// TwinCAT 3 PLC project MasterController
// ProgramVersion: 3.1.4024.0
// libraries:
//   Tc2_EtherCAT, * (Beckhoff Automation GmbH)
//   Tc2_Math, * (Beckhoff Automation GmbH)
//   Tc2_Standard, * (Beckhoff Automation GmbH)
//   Tc2_System, * (Beckhoff Automation GmbH)
//   Tc2_Utilities, * (Beckhoff Automation GmbH)
//   Tc3_Module, * (Beckhoff Automation GmbH)
// project tree:
//   AgiMaths/Frames/ DHTrans.TcPOU (not stored), invFrame.TcPOU (not stored), rotX.TcPOU (not stored), rotY.TcPOU (not stored), rotZ.TcPOU (not stored), transform.TcPOU (not stored)
//   AgiMaths/MatrixLib/ angAxis2Rot.TcPOU (not stored), cross.TcPOU (not stored), Det5.TcPOU (not stored), Det6.TcPOU (not stored), Det7.TcPOU (not stored), invMat6.TcPOU (not stored), invMat6Old.TcPOU (not stored), invMat3.TcPOU (not stored), invMat7.TcPOU (not stored), Mat3T.TcPOU (not stored), matAdd.TcPOU (not stored), matMultiNum.TcPOU (not stored), matMultiply.TcPOU (not stored), matMultiVec.TcPOU (not stored), matSelfAdd.TcPOU (not stored), matSelfSub.TcPOU (not stored), matSub.TcPOU (not stored), matTranspose.TcPOU (not stored), rot2AngAxis.TcPOU (not stored), norm.TcPOU (not stored), normalize.TcPOU (not stored), vecAdd.TcPOU (not stored), vecDot.TcPOU (not stored), vecMultiNum.TcPOU (not stored), vecSelfAdd.TcPOU (not stored), vecSelfMultiNum.TcPOU (not stored), vecSelfSub.TcPOU (not stored), vecSub.TcPOU (not stored)
//   AgiMaths/ sign.TcPOU (not stored), addVec7.TcPOU (not stored), atan2.TcPOU (not stored), cot.TcPOU (not stored)
//   DUTs/Enum/ E_InstruEnergyCtrlWord.TcDUT (not stored), E_InstrumentEnergyType.TcDUT (not stored), E_InstrumentType.TcDUT (not stored), E_MasterArmState.TcDUT, E_MatchedSlaveArmIdx.TcDUT (not stored), E_SlaveArmState.TcDUT (not stored), E_DriverCtrlWord.TcDUT (not stored), E_DriverOPMode.TcDUT (not stored), E_DriverStatusWord.TcDUT (not stored)
//   DUTs/Structure/MasterSlaveCommunication/ ST_MasterStatus.TcDUT (not stored), ST_SlaveStatus.TcDUT (not stored)
//   DUTs/Structure/ ST_EtherCATState.TcDUT (not stored), ST_InstruStatus.TcDUT (not stored), ST_MatchedMasterArmIdx.TcDUT (not stored), ST_ArmCtrlCmds.TcDUT (not stored), ST_MasterInputDataPool.TcDUT (not stored), ST_Frame.TcDUT (not stored)
//   DUTs/Structure/TasksCommunication/ ST_CartUIData.TcDUT (not stored), ST_MasterDynaData.TcDUT (not stored), ST_MasterUIData.TcDUT, ST_CartStatus.TcDUT, ST_MasterJointData.TcDUT (not stored), ST_MotorInputs.TcDUT (not stored), ST_MotorOutputs.TcDUT (not stored), ST_SlaveJointData.TcDUT (not stored), ST_SafetyData.TcDUT (not stored), ST_CartJointData.TcDUT (not stored)
//   DUTs/Structure/UICommunication/ ST_arm_distribution.TcDUT (not stored), ST_ergonCtrlEnable.TcDUT (not stored), ST_ergonomicCtrlData.TcDUT (not stored), ST_instrument_info.TcDUT (not stored), ST_scope_info.TcDUT (not stored)
//   DUTs/Type/ Vec7b.TcDUT (not stored), Mat34.TcDUT (not stored), Mat37.TcDUT (not stored), Mat43.TcDUT (not stored), Mat4d.TcDUT (not stored), Mat5d.TcDUT (not stored), Mat67.TcDUT (not stored), Mat6d.TcDUT (not stored), Mat76.TcDUT (not stored), Mat7d.TcDUT (not stored), Vec4d.TcDUT (not stored), Vec4i.TcDUT (not stored), Vec6i.TcDUT (not stored), Vec4b.TcDUT (not stored), Vec7di.TcDUT (not stored), Vec8d.TcDUT (not stored), Mat3d.TcDUT (not stored), Vec3d.TcDUT (not stored), Vec6d.TcDUT (not stored), Vec7d.TcDUT (not stored), Vec7i.TcDUT (not stored)
//   FBs_Auxiliary/ FB_GripAngleCalc.TcPOU (not stored), FB_HandClutchCheck.TcPOU (not stored), FB_IOCheck.TcPOU (not stored), FB_RiseEdgeCheck.TcPOU (not stored), FB_IOToggleCheck.TcPOU (not stored), FB_MSCtrlTriggerCheck.TcPOU (not stored), FB_slaveConnectionCheck.TcPOU (not stored), FB_TON.TcPOU (not stored)
//   FBs_BasicControllers/ FB_boundaryForceFeedback.TcPOU (not stored), FB_PID.TcPOU (not stored), FB_RedunJntControl.TcPOU
//   FBs_Observer/ FB_JntInertia.TcPOU (not stored), FB_JntObserver.TcPOU (not stored)
//   FBs_RobotDynamics/ FB_MasterDynamic.TcPOU (not stored), FB_MasterFriciton.TcPOU, FB_MasterGravity.TcPOU (not stored)
//   FBs_Robots/ FB_ArmJoint.TcPOU, FB_CartJoint.TcPOU, FB_JointBase.TcPOU, FB_MasterCart.TcPOU, FB_MasterArm.TcPOU, FB_MasterRobot.TcPOU
//   FBs_StateControllers/ FB_EndoscopeController.TcPOU (not stored), FB_StateCtrlClutch.TcPOU (not stored), FB_StateCtrlEndoscope.TcPOU (not stored), FB_StateCtrlCart.TcPOU (not stored), FB_StateCtrlDisable.TcPOU, FB_StateCtrlGraBiasCali.TcPOU (not stored), FB_StateCtrlGraCali.TcPOU, FB_StateCtrlMatching.TcPOU, FB_StateCtrlHome.TcPOU, FB_StateCtrlError.TcPOU, FB_StateCtrlPerformance.TcPOU (not stored), FB_StateCtrlReady.TcPOU (not stored), FB_StateCtrlMasterSlave.TcPOU, FB_StateCtrlTest.TcPOU, FB_StateCtrlInit.TcPOU, FB_StateCtrlStandBy.TcPOU (not stored), FB_MasterArmCtrlBase.TcPOU, I_MasterArmCtrl.TcIO (not stored)
//   FBs_TrajectoryPlanning/ FB_BasicDoubleS.TcPOU (not stored), FB_trajBase.TcPOU (not stored), FB_TrajMoveJ.TcPOU (not stored), linear_trajectory_with_quintic_polynomial_blends.TcPOU (not stored), quintic_spline_curve.TcPOU (not stored), Quintic_spline_curve_factor.TcPOU (not stored), TrapezoIDal_velocity_trajectory.TcPOU (not stored)
//   FBs_TrajectoryPlanning/OTG/ FB_secOrdTrajFilter.TcPOU (not stored), FB_thirdOrdTrajFilter.TcPOU (not stored)
//   FBs_Filters/ FB_LowPassFilter.TcPOU (not stored)
//   GVLs/Arms/ GVL_ArmDynamics.TcGVL, GVL_ArmJointCaliData.TcGVL, GVL_ArmKinematic.TcGVL, GVL_ControlParameters.TcGVL, GVL_ArmJointParameters.TcGVL
//   GVLs/Cart/ GVL_CartJointCaliData.TcGVL, GVL_CartJointParameters.TcGVL
//   GVLs/Configs/Robot3/ GVL_ArmDynamics_3.TcGVL, GVL_ArmJointCaliData_3.TcGVL, GVL_CartJointCaliData_3.TcGVL (not stored)
//   GVLs/Configs/Robot4/ GVL_ArmDynamics_4.TcGVL (not stored), GVL_ArmJointCaliData_4.TcGVL (not stored), GVL_CartJointCaliData_4_1.TcGVL (not stored)
//   GVLs/Configs/Robot5/ GVL_ArmDynamics_5.TcGVL (not stored), GVL_ArmJointCaliData_5.TcGVL (not stored), GVL_CartJointCaliData_5.TcGVL (not stored)
//   GVLs/Configs/Robot6/ GVL_ArmDynamics_6.TcGVL (not stored), GVL_ArmJointCaliData_6.TcGVL (not stored), GVL_CartJointCaliData_6.TcGVL (not stored)
//   GVLs/ GVL_interactUI.TcGVL, GVL_MathDefine.TcGVL (not stored), GVL_SafetyParameters.TcGVL, GVL_SystemParameters.TcGVL
//   Mains/ CartControl.TcPOU (not stored), SafetyCheck.TcPOU (not stored), MasterArmControl.TcPOU, RobotDynamics.TcPOU
//   SafetyCheck/ ASSERT.TcPOU (not stored), Fb_dataRecord.TcPOU (not stored), FB_EtherCATCheck.TcPOU (not stored), Fb_SafetyCheck.TcPOU, FB_Writer.TcPOU (not stored)
//   SafetyCheck/safetyCheckDUT/ checkDelay.TcDUT (not stored), checkDelayTime.TcDUT, checkInputVariable.TcDUT (not stored), checkPermit.TcDUT (not stored), ST_Buffer.TcDUT (not stored), T_Buffer.TcDUT (not stored)
//   Sandbox/ FB_CartCheck.TcPOU (not stored), FB_MasterArmCheck.TcPOU (not stored), FB_RedunJntControl_bak2.TcPOU (not stored), FB_RedunJntControl_bak.TcPOU (not stored)
//   / TaskArmControl.TcTTO (not stored), TaskCartControl.TcTTO (not stored), TaskDynamic.TcTTO (not stored), TaskSafetyCheck.TcTTO (not stored)
// real-time tasks:
//   TASK TaskArmControl: cycle T#250us, priority 1, ADS port 350
//   TASK TaskDynamic: cycle T#1ms, priority 2, ADS port 351
//   TASK TaskSafetyCheck: cycle T#1ms, priority 5, ADS port 352
//   TASK TaskCartControl: cycle T#1ms, priority 4, ADS port 353
// I/O:
//   DEVICE RightArm (EtherCAT), AmsNetId 192.168.0.10.9.1
//     Term 19 (EK1100) [EK1100 EtherCAT Coupler (2A E-Bus)]
//       Term 20 (EL6070) [EL6070 1Ch. Licensing-Terminal]
//       Term 21 (EL1008) [EL1008 8Ch. Dig. Input 24V, 3ms]
//       Term 22 (EL1008) [EL1008 8Ch. Dig. Input 24V, 3ms]
//       Term 23 (EL1008) [EL1008 8Ch. Dig. Input 24V, 3ms]
//       Term 24 (EL2008-0015) [EL2008-0015 8K. Dig. Ausgang 24V DC, 0.35A, nicht kurzschlussfest]
//       Term 25 (EK1122) [EK1122 2 port EtherCAT junction]
//         CartArmSet [AX58200_MotorControl_1axis]
//         CartMonitorLift [AX58200_MotorControl_1axis]
//         CartPedal [AX58200_MotorControl_1axis]
//         CartMonitorRotate [AX58200_MotorControl_1axis]
//     Joint1 [AX58200_MotorControl_1axis]
//     Joint2 [AX58200_MotorControl_1axis]
//     Joint3 [AX58200_MotorControl_1axis]
//     Joint4 [AX58200_MotorControl_1axis]
//     Joint5 [AX58200_MotorControl_1axis]
//     Joint6 [AX58200_MotorControl_1axis]
//     Joint7 [AX58200_MotorControl_1axis]
//   DEVICE LeftArm (EtherCAT), AmsNetId 192.168.0.10.4.1
//     Joint1 [AX58200_MotorControl_1axis]
//     Joint2 [AX58200_MotorControl_1axis]
//     Joint3 [AX58200_MotorControl_1axis]
//     Joint4 [AX58200_MotorControl_1axis]
//     Joint5 [AX58200_MotorControl_1axis]
//     Joint6 [AX58200_MotorControl_1axis]
//     Joint7 [AX58200_MotorControl_1axis]
//   DEVICE MSCommunication (EtherCAT), AmsNetId 192.168.0.10.7.1
//     Box 45 (AX58200_MotorControl) [AX58200_MotorControl2021.9.13]
//     Box 46 (EL6695-0002) [EL6695 EtherCAT Bridge terminal (Secondary)]
// variable links:
//   MasterController/MasterController Instance <-> LeftArm (EtherCAT)/Joint1
//     TaskArmControl Inputs/MasterArmControl.m_masterRobot.m_masterArms[1].m_joints[1].m_motorInputs/m_current <-> TxPdoMappingCspCsv/Torque actual value
//     TaskArmControl Inputs/MasterArmControl.m_masterRobot.m_masterArms[1].m_joints[1].m_motorInputs/m_driverError <-> TxPdoMappingCspCsv/digital input
//     TaskArmControl Inputs/MasterArmControl.m_masterRobot.m_masterArms[1].m_joints[1].m_motorInputs/m_linkEncoder <-> TxPdoMappingCspCsv/ENC2
//     TaskArmControl Inputs/MasterArmControl.m_masterRobot.m_masterArms[1].m_joints[1].m_motorInputs/m_motorEncoder <-> TxPdoMappingCspCsv/Position actual value
//     TaskArmControl Inputs/MasterArmControl.m_masterRobot.m_masterArms[1].m_joints[1].m_motorInputs/m_statusWord <-> TxPdoMappingCspCsv/Statusword
//     TaskArmControl Outputs/MasterArmControl.m_masterRobot.m_masterArms[1].m_joints[1].m_motorOutputs/m_cmdCurrent <-> RxPdoMappingCspCsv/Target torque
//     TaskArmControl Outputs/MasterArmControl.m_masterRobot.m_masterArms[1].m_joints[1].m_motorOutputs/m_cmdMotorEncoder <-> RxPdoMappingCspCsv/Target position
//     TaskArmControl Outputs/MasterArmControl.m_masterRobot.m_masterArms[1].m_joints[1].m_motorOutputs/m_controlWord <-> RxPdoMappingCspCsv/Controlword
//     TaskArmControl Outputs/MasterArmControl.m_masterRobot.m_masterArms[1].m_joints[1].m_motorOutputs/m_opMode <-> RxPdoMappingCspCsv/Modes of operation
//   MasterController/MasterController Instance <-> LeftArm (EtherCAT)/Joint2
//     TaskArmControl Inputs/MasterArmControl.m_masterRobot.m_masterArms[1].m_joints[2].m_motorInputs/m_current <-> TxPdoMappingCspCsv/Torque actual value
//     TaskArmControl Inputs/MasterArmControl.m_masterRobot.m_masterArms[1].m_joints[2].m_motorInputs/m_driverError <-> TxPdoMappingCspCsv/digital input
//     TaskArmControl Inputs/MasterArmControl.m_masterRobot.m_masterArms[1].m_joints[2].m_motorInputs/m_linkEncoder <-> TxPdoMappingCspCsv/ENC2
//     TaskArmControl Inputs/MasterArmControl.m_masterRobot.m_masterArms[1].m_joints[2].m_motorInputs/m_motorEncoder <-> TxPdoMappingCspCsv/Position actual value
//     TaskArmControl Inputs/MasterArmControl.m_masterRobot.m_masterArms[1].m_joints[2].m_motorInputs/m_statusWord <-> TxPdoMappingCspCsv/Statusword
//     TaskArmControl Outputs/MasterArmControl.m_masterRobot.m_masterArms[1].m_joints[2].m_motorOutputs/m_cmdCurrent <-> RxPdoMappingCspCsv/Target torque
//     TaskArmControl Outputs/MasterArmControl.m_masterRobot.m_masterArms[1].m_joints[2].m_motorOutputs/m_cmdMotorEncoder <-> RxPdoMappingCspCsv/Target position
//     TaskArmControl Outputs/MasterArmControl.m_masterRobot.m_masterArms[1].m_joints[2].m_motorOutputs/m_controlWord <-> RxPdoMappingCspCsv/Controlword
//     TaskArmControl Outputs/MasterArmControl.m_masterRobot.m_masterArms[1].m_joints[2].m_motorOutputs/m_opMode <-> RxPdoMappingCspCsv/Modes of operation
//   MasterController/MasterController Instance <-> LeftArm (EtherCAT)/Joint3
//     TaskArmControl Inputs/MasterArmControl.m_masterRobot.m_masterArms[1].m_joints[3].m_motorInputs/m_current <-> TxPdoMappingCspCsv/Torque actual value
//     TaskArmControl Inputs/MasterArmControl.m_masterRobot.m_masterArms[1].m_joints[3].m_motorInputs/m_driverError <-> TxPdoMappingCspCsv/digital input
//     TaskArmControl Inputs/MasterArmControl.m_masterRobot.m_masterArms[1].m_joints[3].m_motorInputs/m_linkEncoder <-> TxPdoMappingCspCsv/ENC2
//     TaskArmControl Inputs/MasterArmControl.m_masterRobot.m_masterArms[1].m_joints[3].m_motorInputs/m_motorEncoder <-> TxPdoMappingCspCsv/Position actual value
//     TaskArmControl Inputs/MasterArmControl.m_masterRobot.m_masterArms[1].m_joints[3].m_motorInputs/m_statusWord <-> TxPdoMappingCspCsv/Statusword
//     TaskArmControl Outputs/MasterArmControl.m_masterRobot.m_masterArms[1].m_joints[3].m_motorOutputs/m_cmdCurrent <-> RxPdoMappingCspCsv/Target torque
//     TaskArmControl Outputs/MasterArmControl.m_masterRobot.m_masterArms[1].m_joints[3].m_motorOutputs/m_cmdMotorEncoder <-> RxPdoMappingCspCsv/Target position
//     TaskArmControl Outputs/MasterArmControl.m_masterRobot.m_masterArms[1].m_joints[3].m_motorOutputs/m_controlWord <-> RxPdoMappingCspCsv/Controlword
//     TaskArmControl Outputs/MasterArmControl.m_masterRobot.m_masterArms[1].m_joints[3].m_motorOutputs/m_opMode <-> RxPdoMappingCspCsv/Modes of operation
//   MasterController/MasterController Instance <-> LeftArm (EtherCAT)/Joint4
//     TaskArmControl Inputs/MasterArmControl.m_masterRobot.m_masterArms[1].m_joints[4].m_motorInputs/m_current <-> TxPdoMappingCspCsv/Torque actual value
//     TaskArmControl Inputs/MasterArmControl.m_masterRobot.m_masterArms[1].m_joints[4].m_motorInputs/m_driverError <-> TxPdoMappingCspCsv/digital input
//     TaskArmControl Inputs/MasterArmControl.m_masterRobot.m_masterArms[1].m_joints[4].m_motorInputs/m_motorEncoder <-> TxPdoMappingCspCsv/Position actual value
//     TaskArmControl Inputs/MasterArmControl.m_masterRobot.m_masterArms[1].m_joints[4].m_motorInputs/m_statusWord <-> TxPdoMappingCspCsv/Statusword
//     TaskArmControl Outputs/MasterArmControl.m_masterRobot.m_masterArms[1].m_joints[4].m_motorOutputs/m_cmdCurrent <-> RxPdoMappingCspCsv/Target torque
//     TaskArmControl Outputs/MasterArmControl.m_masterRobot.m_masterArms[1].m_joints[4].m_motorOutputs/m_cmdMotorEncoder <-> RxPdoMappingCspCsv/Target position
//     TaskArmControl Outputs/MasterArmControl.m_masterRobot.m_masterArms[1].m_joints[4].m_motorOutputs/m_controlWord <-> RxPdoMappingCspCsv/Controlword
//     TaskArmControl Outputs/MasterArmControl.m_masterRobot.m_masterArms[1].m_joints[4].m_motorOutputs/m_opMode <-> RxPdoMappingCspCsv/Modes of operation
//   MasterController/MasterController Instance <-> LeftArm (EtherCAT)/Joint5
//     TaskArmControl Inputs/MasterArmControl.m_masterRobot.m_masterArms[1].m_joints[4].m_motorInputs/m_linkEncoder <-> TxPdoMappingCspCsv/Velocity actual value
//     TaskArmControl Inputs/MasterArmControl.m_masterRobot.m_masterArms[1].m_joints[5].m_motorInputs/m_current <-> TxPdoMappingCspCsv/Torque actual value
//     TaskArmControl Inputs/MasterArmControl.m_masterRobot.m_masterArms[1].m_joints[5].m_motorInputs/m_driverError <-> TxPdoMappingCspCsv/digital input
//     TaskArmControl Inputs/MasterArmControl.m_masterRobot.m_masterArms[1].m_joints[5].m_motorInputs/m_linkEncoder <-> TxPdoMappingCspCsv/ENC2
//     TaskArmControl Inputs/MasterArmControl.m_masterRobot.m_masterArms[1].m_joints[5].m_motorInputs/m_motorEncoder <-> TxPdoMappingCspCsv/Position actual value
//     TaskArmControl Inputs/MasterArmControl.m_masterRobot.m_masterArms[1].m_joints[5].m_motorInputs/m_statusWord <-> TxPdoMappingCspCsv/Statusword
//     TaskArmControl Outputs/MasterArmControl.m_masterRobot.m_masterArms[1].m_joints[5].m_motorOutputs/m_cmdCurrent <-> RxPdoMappingCspCsv/Target torque
//     TaskArmControl Outputs/MasterArmControl.m_masterRobot.m_masterArms[1].m_joints[5].m_motorOutputs/m_cmdMotorEncoder <-> RxPdoMappingCspCsv/Target position
//     TaskArmControl Outputs/MasterArmControl.m_masterRobot.m_masterArms[1].m_joints[5].m_motorOutputs/m_controlWord <-> RxPdoMappingCspCsv/Controlword
//     TaskArmControl Outputs/MasterArmControl.m_masterRobot.m_masterArms[1].m_joints[5].m_motorOutputs/m_opMode <-> RxPdoMappingCspCsv/Modes of operation
//   MasterController/MasterController Instance <-> LeftArm (EtherCAT)/Joint6
//     TaskArmControl Inputs/MasterArmControl.m_masterRobot.m_masterArms[1].m_joints[6].m_motorInputs/m_current <-> TxPdoMappingCspCsv/Torque actual value
//     TaskArmControl Inputs/MasterArmControl.m_masterRobot.m_masterArms[1].m_joints[6].m_motorInputs/m_driverError <-> TxPdoMappingCspCsv/digital input
//     TaskArmControl Inputs/MasterArmControl.m_masterRobot.m_masterArms[1].m_joints[6].m_motorInputs/m_linkEncoder <-> TxPdoMappingCspCsv/ENC2
//     TaskArmControl Inputs/MasterArmControl.m_masterRobot.m_masterArms[1].m_joints[6].m_motorInputs/m_motorEncoder <-> TxPdoMappingCspCsv/Position actual value
//     TaskArmControl Inputs/MasterArmControl.m_masterRobot.m_masterArms[1].m_joints[6].m_motorInputs/m_statusWord <-> TxPdoMappingCspCsv/Statusword
//     TaskArmControl Outputs/MasterArmControl.m_masterRobot.m_masterArms[1].m_joints[6].m_motorOutputs/m_cmdCurrent <-> RxPdoMappingCspCsv/Target torque
//     TaskArmControl Outputs/MasterArmControl.m_masterRobot.m_masterArms[1].m_joints[6].m_motorOutputs/m_cmdMotorEncoder <-> RxPdoMappingCspCsv/Target position
//     TaskArmControl Outputs/MasterArmControl.m_masterRobot.m_masterArms[1].m_joints[6].m_motorOutputs/m_controlWord <-> RxPdoMappingCspCsv/Controlword
//     TaskArmControl Outputs/MasterArmControl.m_masterRobot.m_masterArms[1].m_joints[6].m_motorOutputs/m_opMode <-> RxPdoMappingCspCsv/Modes of operation
//   MasterController/MasterController Instance <-> LeftArm (EtherCAT)/Joint7
//     TaskArmControl Inputs/MasterArmControl.m_masterRobot.m_masterArms[1].m_gripHallSensorIO <-> TxPdoMappingCspCsv/analog input
//     TaskArmControl Inputs/MasterArmControl.m_masterRobot.m_masterArms[1].m_handClutchIO <-> TxPdoMappingCspCsv/digital input
//     TaskArmControl Inputs/MasterArmControl.m_masterRobot.m_masterArms[1].m_joints[7].m_motorInputs/m_current <-> TxPdoMappingCspCsv/Torque actual value
//     TaskArmControl Inputs/MasterArmControl.m_masterRobot.m_masterArms[1].m_joints[7].m_motorInputs/m_linkEncoder <-> TxPdoMappingCspCsv/ENC2
//     TaskArmControl Inputs/MasterArmControl.m_masterRobot.m_masterArms[1].m_joints[7].m_motorInputs/m_motorEncoder <-> TxPdoMappingCspCsv/Position actual value
//     TaskArmControl Inputs/MasterArmControl.m_masterRobot.m_masterArms[1].m_joints[7].m_motorInputs/m_statusWord <-> TxPdoMappingCspCsv/Statusword
//     TaskArmControl Outputs/MasterArmControl.m_masterRobot.m_masterArms[1].m_joints[7].m_motorOutputs/m_cmdCurrent <-> RxPdoMappingCspCsv/Target torque
//     TaskArmControl Outputs/MasterArmControl.m_masterRobot.m_masterArms[1].m_joints[7].m_motorOutputs/m_cmdMotorEncoder <-> RxPdoMappingCspCsv/Target position
//     TaskArmControl Outputs/MasterArmControl.m_masterRobot.m_masterArms[1].m_joints[7].m_motorOutputs/m_controlWord <-> RxPdoMappingCspCsv/Controlword
//     TaskArmControl Outputs/MasterArmControl.m_masterRobot.m_masterArms[1].m_joints[7].m_motorOutputs/m_opMode <-> RxPdoMappingCspCsv/Modes of operation
//   MasterController/MasterController Instance <-> MSCommunication (EtherCAT)/Box 45 (AX58200_MotorControl)
//     TaskCartControl Outputs/CartControl.m_masterCart.m_elecKnifeCtrlWord <-> RxPdoMappingCspCsv/Target velocity
//   MasterController/MasterController Instance <-> MSCommunication (EtherCAT)/Box 46 (EL6695-0002)
//     TaskArmControl Inputs/MasterArmControl.m_slaveRobotData <-> IO Inputs/SlaveRobotData
//     TaskArmControl Outputs/MasterArmControl.m_masterRobotData <-> IO Outputs/MasterRobotData
//   MasterController/MasterController Instance <-> RightArm (EtherCAT)/Joint1
//     TaskArmControl Inputs/MasterArmControl.m_masterRobot.m_masterArms[2].m_joints[1].m_motorInputs/m_current <-> TxPdoMappingCspCsv/Torque actual value
//     TaskArmControl Inputs/MasterArmControl.m_masterRobot.m_masterArms[2].m_joints[1].m_motorInputs/m_driverError <-> TxPdoMappingCspCsv/digital input
//     TaskArmControl Inputs/MasterArmControl.m_masterRobot.m_masterArms[2].m_joints[1].m_motorInputs/m_linkEncoder <-> TxPdoMappingCspCsv/ENC2
//     TaskArmControl Inputs/MasterArmControl.m_masterRobot.m_masterArms[2].m_joints[1].m_motorInputs/m_motorEncoder <-> TxPdoMappingCspCsv/Position actual value
//     TaskArmControl Inputs/MasterArmControl.m_masterRobot.m_masterArms[2].m_joints[1].m_motorInputs/m_statusWord <-> TxPdoMappingCspCsv/Statusword
//     TaskArmControl Outputs/MasterArmControl.m_masterRobot.m_masterArms[2].m_joints[1].m_motorOutputs/m_cmdCurrent <-> RxPdoMappingCspCsv/Target torque
//     TaskArmControl Outputs/MasterArmControl.m_masterRobot.m_masterArms[2].m_joints[1].m_motorOutputs/m_cmdMotorEncoder <-> RxPdoMappingCspCsv/Target position
//     TaskArmControl Outputs/MasterArmControl.m_masterRobot.m_masterArms[2].m_joints[1].m_motorOutputs/m_controlWord <-> RxPdoMappingCspCsv/Controlword
//     TaskArmControl Outputs/MasterArmControl.m_masterRobot.m_masterArms[2].m_joints[1].m_motorOutputs/m_opMode <-> RxPdoMappingCspCsv/Modes of operation
//   MasterController/MasterController Instance <-> RightArm (EtherCAT)/Joint2
//     TaskArmControl Inputs/MasterArmControl.m_masterRobot.m_masterArms[2].m_joints[2].m_motorInputs/m_current <-> TxPdoMappingCspCsv/Torque actual value
//     TaskArmControl Inputs/MasterArmControl.m_masterRobot.m_masterArms[2].m_joints[2].m_motorInputs/m_driverError <-> TxPdoMappingCspCsv/digital input
//     TaskArmControl Inputs/MasterArmControl.m_masterRobot.m_masterArms[2].m_joints[2].m_motorInputs/m_linkEncoder <-> TxPdoMappingCspCsv/ENC2
//     TaskArmControl Inputs/MasterArmControl.m_masterRobot.m_masterArms[2].m_joints[2].m_motorInputs/m_motorEncoder <-> TxPdoMappingCspCsv/Position actual value
//     TaskArmControl Inputs/MasterArmControl.m_masterRobot.m_masterArms[2].m_joints[2].m_motorInputs/m_statusWord <-> TxPdoMappingCspCsv/Statusword
//     TaskArmControl Outputs/MasterArmControl.m_masterRobot.m_masterArms[2].m_joints[2].m_motorOutputs/m_cmdCurrent <-> RxPdoMappingCspCsv/Target torque
//     TaskArmControl Outputs/MasterArmControl.m_masterRobot.m_masterArms[2].m_joints[2].m_motorOutputs/m_cmdMotorEncoder <-> RxPdoMappingCspCsv/Target position
//     TaskArmControl Outputs/MasterArmControl.m_masterRobot.m_masterArms[2].m_joints[2].m_motorOutputs/m_controlWord <-> RxPdoMappingCspCsv/Controlword
//     TaskArmControl Outputs/MasterArmControl.m_masterRobot.m_masterArms[2].m_joints[2].m_motorOutputs/m_opMode <-> RxPdoMappingCspCsv/Modes of operation
//   MasterController/MasterController Instance <-> RightArm (EtherCAT)/Joint3
//     TaskArmControl Inputs/MasterArmControl.m_masterRobot.m_masterArms[2].m_joints[3].m_motorInputs/m_current <-> TxPdoMappingCspCsv/Torque actual value
//     TaskArmControl Inputs/MasterArmControl.m_masterRobot.m_masterArms[2].m_joints[3].m_motorInputs/m_driverError <-> TxPdoMappingCspCsv/digital input
//     TaskArmControl Inputs/MasterArmControl.m_masterRobot.m_masterArms[2].m_joints[3].m_motorInputs/m_linkEncoder <-> TxPdoMappingCspCsv/ENC2
//     TaskArmControl Inputs/MasterArmControl.m_masterRobot.m_masterArms[2].m_joints[3].m_motorInputs/m_motorEncoder <-> TxPdoMappingCspCsv/Position actual value
//     TaskArmControl Inputs/MasterArmControl.m_masterRobot.m_masterArms[2].m_joints[3].m_motorInputs/m_statusWord <-> TxPdoMappingCspCsv/Statusword
//     TaskArmControl Outputs/MasterArmControl.m_masterRobot.m_masterArms[2].m_joints[3].m_motorOutputs/m_cmdCurrent <-> RxPdoMappingCspCsv/Target torque
//     TaskArmControl Outputs/MasterArmControl.m_masterRobot.m_masterArms[2].m_joints[3].m_motorOutputs/m_cmdMotorEncoder <-> RxPdoMappingCspCsv/Target position
//     TaskArmControl Outputs/MasterArmControl.m_masterRobot.m_masterArms[2].m_joints[3].m_motorOutputs/m_controlWord <-> RxPdoMappingCspCsv/Controlword
//     TaskArmControl Outputs/MasterArmControl.m_masterRobot.m_masterArms[2].m_joints[3].m_motorOutputs/m_opMode <-> RxPdoMappingCspCsv/Modes of operation
//   MasterController/MasterController Instance <-> RightArm (EtherCAT)/Joint4
//     TaskArmControl Inputs/MasterArmControl.m_masterRobot.m_masterArms[2].m_joints[4].m_motorInputs/m_current <-> TxPdoMappingCspCsv/Torque actual value
//     TaskArmControl Inputs/MasterArmControl.m_masterRobot.m_masterArms[2].m_joints[4].m_motorInputs/m_driverError <-> TxPdoMappingCspCsv/digital input
//     TaskArmControl Inputs/MasterArmControl.m_masterRobot.m_masterArms[2].m_joints[4].m_motorInputs/m_motorEncoder <-> TxPdoMappingCspCsv/Position actual value
//     TaskArmControl Inputs/MasterArmControl.m_masterRobot.m_masterArms[2].m_joints[4].m_motorInputs/m_statusWord <-> TxPdoMappingCspCsv/Statusword
//     TaskArmControl Outputs/MasterArmControl.m_masterRobot.m_masterArms[2].m_joints[4].m_motorOutputs/m_cmdCurrent <-> RxPdoMappingCspCsv/Target torque
//     TaskArmControl Outputs/MasterArmControl.m_masterRobot.m_masterArms[2].m_joints[4].m_motorOutputs/m_cmdMotorEncoder <-> RxPdoMappingCspCsv/Target position
//     TaskArmControl Outputs/MasterArmControl.m_masterRobot.m_masterArms[2].m_joints[4].m_motorOutputs/m_controlWord <-> RxPdoMappingCspCsv/Controlword
//     TaskArmControl Outputs/MasterArmControl.m_masterRobot.m_masterArms[2].m_joints[4].m_motorOutputs/m_opMode <-> RxPdoMappingCspCsv/Modes of operation
//   MasterController/MasterController Instance <-> RightArm (EtherCAT)/Joint5
//     TaskArmControl Inputs/MasterArmControl.m_masterRobot.m_masterArms[2].m_joints[4].m_motorInputs/m_linkEncoder <-> TxPdoMappingCspCsv/Velocity actual value
//     TaskArmControl Inputs/MasterArmControl.m_masterRobot.m_masterArms[2].m_joints[5].m_motorInputs/m_current <-> TxPdoMappingCspCsv/Torque actual value
//     TaskArmControl Inputs/MasterArmControl.m_masterRobot.m_masterArms[2].m_joints[5].m_motorInputs/m_driverError <-> TxPdoMappingCspCsv/digital input
//     TaskArmControl Inputs/MasterArmControl.m_masterRobot.m_masterArms[2].m_joints[5].m_motorInputs/m_linkEncoder <-> TxPdoMappingCspCsv/ENC2
//     TaskArmControl Inputs/MasterArmControl.m_masterRobot.m_masterArms[2].m_joints[5].m_motorInputs/m_motorEncoder <-> TxPdoMappingCspCsv/Position actual value
//     TaskArmControl Inputs/MasterArmControl.m_masterRobot.m_masterArms[2].m_joints[5].m_motorInputs/m_statusWord <-> TxPdoMappingCspCsv/Statusword
//     TaskArmControl Outputs/MasterArmControl.m_masterRobot.m_masterArms[2].m_joints[5].m_motorOutputs/m_cmdCurrent <-> RxPdoMappingCspCsv/Target torque
//     TaskArmControl Outputs/MasterArmControl.m_masterRobot.m_masterArms[2].m_joints[5].m_motorOutputs/m_cmdMotorEncoder <-> RxPdoMappingCspCsv/Target position
//     TaskArmControl Outputs/MasterArmControl.m_masterRobot.m_masterArms[2].m_joints[5].m_motorOutputs/m_controlWord <-> RxPdoMappingCspCsv/Controlword
//     TaskArmControl Outputs/MasterArmControl.m_masterRobot.m_masterArms[2].m_joints[5].m_motorOutputs/m_opMode <-> RxPdoMappingCspCsv/Modes of operation
//   MasterController/MasterController Instance <-> RightArm (EtherCAT)/Joint6
//     TaskArmControl Inputs/MasterArmControl.m_masterRobot.m_masterArms[2].m_joints[6].m_motorInputs/m_current <-> TxPdoMappingCspCsv/Torque actual value
//     TaskArmControl Inputs/MasterArmControl.m_masterRobot.m_masterArms[2].m_joints[6].m_motorInputs/m_driverError <-> TxPdoMappingCspCsv/digital input
//     TaskArmControl Inputs/MasterArmControl.m_masterRobot.m_masterArms[2].m_joints[6].m_motorInputs/m_linkEncoder <-> TxPdoMappingCspCsv/ENC2
//     TaskArmControl Inputs/MasterArmControl.m_masterRobot.m_masterArms[2].m_joints[6].m_motorInputs/m_motorEncoder <-> TxPdoMappingCspCsv/Position actual value
//     TaskArmControl Inputs/MasterArmControl.m_masterRobot.m_masterArms[2].m_joints[6].m_motorInputs/m_statusWord <-> TxPdoMappingCspCsv/Statusword
//     TaskArmControl Outputs/MasterArmControl.m_masterRobot.m_masterArms[2].m_joints[6].m_motorOutputs/m_cmdCurrent <-> RxPdoMappingCspCsv/Target torque
//     TaskArmControl Outputs/MasterArmControl.m_masterRobot.m_masterArms[2].m_joints[6].m_motorOutputs/m_cmdMotorEncoder <-> RxPdoMappingCspCsv/Target position
//     TaskArmControl Outputs/MasterArmControl.m_masterRobot.m_masterArms[2].m_joints[6].m_motorOutputs/m_controlWord <-> RxPdoMappingCspCsv/Controlword
//     TaskArmControl Outputs/MasterArmControl.m_masterRobot.m_masterArms[2].m_joints[6].m_motorOutputs/m_opMode <-> RxPdoMappingCspCsv/Modes of operation
//   MasterController/MasterController Instance <-> RightArm (EtherCAT)/Joint7
//     TaskArmControl Inputs/MasterArmControl.m_masterRobot.m_masterArms[2].m_gripHallSensorIO <-> TxPdoMappingCspCsv/analog input
//     TaskArmControl Inputs/MasterArmControl.m_masterRobot.m_masterArms[2].m_handClutchIO <-> TxPdoMappingCspCsv/digital input
//     TaskArmControl Inputs/MasterArmControl.m_masterRobot.m_masterArms[2].m_joints[7].m_motorInputs/m_current <-> TxPdoMappingCspCsv/Torque actual value
//     TaskArmControl Inputs/MasterArmControl.m_masterRobot.m_masterArms[2].m_joints[7].m_motorInputs/m_linkEncoder <-> TxPdoMappingCspCsv/ENC2
//     TaskArmControl Inputs/MasterArmControl.m_masterRobot.m_masterArms[2].m_joints[7].m_motorInputs/m_motorEncoder <-> TxPdoMappingCspCsv/Position actual value
//     TaskArmControl Inputs/MasterArmControl.m_masterRobot.m_masterArms[2].m_joints[7].m_motorInputs/m_statusWord <-> TxPdoMappingCspCsv/Statusword
//     TaskArmControl Outputs/MasterArmControl.m_masterRobot.m_masterArms[2].m_joints[7].m_motorOutputs/m_cmdCurrent <-> RxPdoMappingCspCsv/Target torque
//     TaskArmControl Outputs/MasterArmControl.m_masterRobot.m_masterArms[2].m_joints[7].m_motorOutputs/m_cmdMotorEncoder <-> RxPdoMappingCspCsv/Target position
//     TaskArmControl Outputs/MasterArmControl.m_masterRobot.m_masterArms[2].m_joints[7].m_motorOutputs/m_controlWord <-> RxPdoMappingCspCsv/Controlword
//     TaskArmControl Outputs/MasterArmControl.m_masterRobot.m_masterArms[2].m_joints[7].m_motorOutputs/m_opMode <-> RxPdoMappingCspCsv/Modes of operation
//   MasterController/MasterController Instance <-> RightArm (EtherCAT)/Term 19 (EK1100)/Term 21 (EL1008)
//     TaskArmControl Inputs/SafetyCheck.m_stopButton <-> Channel 1/CartControl.m_masterCart.m_stopButton
//     TaskCartControl Inputs/CartControl.m_masterCart.m_armSwitchIO <-> Channel 4/armSwitchIO
//     TaskCartControl Inputs/CartControl.m_masterCart.m_clutchPedalIO <-> Channel 2/CartControl.m_masterCart.m_clutchPedalIO
//     TaskCartControl Inputs/CartControl.m_masterCart.m_electricCoagulLeft <-> Channel 7/Input
//     TaskCartControl Inputs/CartControl.m_masterCart.m_electricCoagulRight <-> Channel 8/Input
//     TaskCartControl Inputs/CartControl.m_masterCart.m_electricCutLeft <-> Channel 5/Input
//     TaskCartControl Inputs/CartControl.m_masterCart.m_electricCutRight <-> Channel 6/Input
//     TaskCartControl Inputs/CartControl.m_masterCart.m_endoScopePedalIO <-> Channel 3/endoscopePedaoIO
//   MasterController/MasterController Instance <-> RightArm (EtherCAT)/Term 19 (EK1100)/Term 22 (EL1008)
//     TaskCartControl Inputs/CartControl.m_masterCart.m_electricCoagulLeftAllow <-> Channel 2/Input
//     TaskCartControl Inputs/CartControl.m_masterCart.m_electricCoagulRightAllow <-> Channel 4/Input
//     TaskCartControl Inputs/CartControl.m_masterCart.m_electricCutLeftAllow <-> Channel 1/Input
//     TaskCartControl Inputs/CartControl.m_masterCart.m_electricCutRightAllow <-> Channel 3/Input
//     TaskCartControl Inputs/CartControl.m_masterCart.m_surgonHeadInIO <-> Channel 5/HeadInIO
//     TaskSafetyCheck Inputs/SafetyCheck.m_cartLockSignalLeft <-> Channel 7/Input
//     TaskSafetyCheck Inputs/SafetyCheck.m_cartLockSignalRight <-> Channel 8/Input
//   MasterController/MasterController Instance <-> RightArm (EtherCAT)/Term 19 (EK1100)/Term 23 (EL1008)
//     TaskCartControl Inputs/CartControl.m_masterCart.m_cartJointCtrlIO[1] <-> Channel 1/monitorUp
//     TaskCartControl Inputs/CartControl.m_masterCart.m_cartJointCtrlIO[2] <-> Channel 2/monitorDown
//     TaskCartControl Inputs/CartControl.m_masterCart.m_cartJointCtrlIO[3] <-> Channel 8/monitorCCW
//     TaskCartControl Inputs/CartControl.m_masterCart.m_cartJointCtrlIO[4] <-> Channel 7/monitorCW
//     TaskCartControl Inputs/CartControl.m_masterCart.m_cartJointCtrlIO[5] <-> Channel 3/armSetUp
//     TaskCartControl Inputs/CartControl.m_masterCart.m_cartJointCtrlIO[6] <-> Channel 4/armSetDown
//     TaskCartControl Inputs/CartControl.m_masterCart.m_cartJointCtrlIO[7] <-> Channel 5/pedalIn
//     TaskCartControl Inputs/CartControl.m_masterCart.m_cartJointCtrlIO[8] <-> Channel 6/pedalOut
//   MasterController/MasterController Instance <-> RightArm (EtherCAT)/Term 19 (EK1100)/Term 25 (EK1122)/CartArmSet
//     TaskCartControl Inputs/CartControl.m_masterCart.m_cartJoints[3].m_motorInputs/m_current <-> TxPdoMappingCspCsv/Torque actual value
//     TaskCartControl Inputs/CartControl.m_masterCart.m_cartJoints[3].m_motorInputs/m_linkEncoder <-> TxPdoMappingCspCsv/ENC2
//     TaskCartControl Inputs/CartControl.m_masterCart.m_cartJoints[3].m_motorInputs/m_motorEncoder <-> TxPdoMappingCspCsv/Position actual value
//     TaskCartControl Inputs/CartControl.m_masterCart.m_cartJoints[3].m_motorInputs/m_statusWord <-> TxPdoMappingCspCsv/Statusword
//     TaskCartControl Outputs/CartControl.m_masterCart.m_cartJoints[3].m_motorOutputs/m_cmdCurrent <-> RxPdoMappingCspCsv/Target torque
//     TaskCartControl Outputs/CartControl.m_masterCart.m_cartJoints[3].m_motorOutputs/m_cmdMotorEncoder <-> RxPdoMappingCspCsv/Target position
//     TaskCartControl Outputs/CartControl.m_masterCart.m_cartJoints[3].m_motorOutputs/m_controlWord <-> RxPdoMappingCspCsv/Controlword
//     TaskCartControl Outputs/CartControl.m_masterCart.m_cartJoints[3].m_motorOutputs/m_opMode <-> RxPdoMappingCspCsv/Modes of operation
//   MasterController/MasterController Instance <-> RightArm (EtherCAT)/Term 19 (EK1100)/Term 25 (EK1122)/CartMonitorLift
//     TaskCartControl Inputs/CartControl.m_masterCart.m_cartJoints[1].m_motorInputs/m_current <-> TxPdoMappingCspCsv/Torque actual value
//     TaskCartControl Inputs/CartControl.m_masterCart.m_cartJoints[1].m_motorInputs/m_linkEncoder <-> TxPdoMappingCspCsv/ENC2
//     TaskCartControl Inputs/CartControl.m_masterCart.m_cartJoints[1].m_motorInputs/m_motorEncoder <-> TxPdoMappingCspCsv/Position actual value
//     TaskCartControl Inputs/CartControl.m_masterCart.m_cartJoints[1].m_motorInputs/m_statusWord <-> TxPdoMappingCspCsv/Statusword
//     TaskCartControl Outputs/CartControl.m_masterCart.m_cartJoints[1].m_motorOutputs/m_cmdCurrent <-> RxPdoMappingCspCsv/Target torque
//     TaskCartControl Outputs/CartControl.m_masterCart.m_cartJoints[1].m_motorOutputs/m_cmdMotorEncoder <-> RxPdoMappingCspCsv/Target position
//     TaskCartControl Outputs/CartControl.m_masterCart.m_cartJoints[1].m_motorOutputs/m_controlWord <-> RxPdoMappingCspCsv/Controlword
//     TaskCartControl Outputs/CartControl.m_masterCart.m_cartJoints[1].m_motorOutputs/m_opMode <-> RxPdoMappingCspCsv/Modes of operation
//   MasterController/MasterController Instance <-> RightArm (EtherCAT)/Term 19 (EK1100)/Term 25 (EK1122)/CartMonitorRotate
//     TaskCartControl Inputs/CartControl.m_masterCart.m_cartJoints[2].m_motorInputs/m_current <-> TxPdoMappingCspCsv/Torque actual value
//     TaskCartControl Inputs/CartControl.m_masterCart.m_cartJoints[2].m_motorInputs/m_linkEncoder <-> TxPdoMappingCspCsv/ENC2
//     TaskCartControl Inputs/CartControl.m_masterCart.m_cartJoints[2].m_motorInputs/m_motorEncoder <-> TxPdoMappingCspCsv/Position actual value
//     TaskCartControl Inputs/CartControl.m_masterCart.m_cartJoints[2].m_motorInputs/m_statusWord <-> TxPdoMappingCspCsv/Statusword
//     TaskCartControl Outputs/CartControl.m_masterCart.m_cartJoints[2].m_motorOutputs/m_cmdCurrent <-> RxPdoMappingCspCsv/Target torque
//     TaskCartControl Outputs/CartControl.m_masterCart.m_cartJoints[2].m_motorOutputs/m_cmdMotorEncoder <-> RxPdoMappingCspCsv/Target position
//     TaskCartControl Outputs/CartControl.m_masterCart.m_cartJoints[2].m_motorOutputs/m_controlWord <-> RxPdoMappingCspCsv/Controlword
//     TaskCartControl Outputs/CartControl.m_masterCart.m_cartJoints[2].m_motorOutputs/m_opMode <-> RxPdoMappingCspCsv/Modes of operation
//   MasterController/MasterController Instance <-> RightArm (EtherCAT)/Term 19 (EK1100)/Term 25 (EK1122)/CartPedal
//     TaskCartControl Inputs/CartControl.m_masterCart.m_cartJoints[4].m_motorInputs/m_current <-> TxPdoMappingCspCsv/Torque actual value
//     TaskCartControl Inputs/CartControl.m_masterCart.m_cartJoints[4].m_motorInputs/m_linkEncoder <-> TxPdoMappingCspCsv/ENC2
//     TaskCartControl Inputs/CartControl.m_masterCart.m_cartJoints[4].m_motorInputs/m_motorEncoder <-> TxPdoMappingCspCsv/Position actual value
//     TaskCartControl Inputs/CartControl.m_masterCart.m_cartJoints[4].m_motorInputs/m_statusWord <-> TxPdoMappingCspCsv/Statusword
//     TaskCartControl Outputs/CartControl.m_masterCart.m_cartJoints[4].m_motorOutputs/m_cmdCurrent <-> RxPdoMappingCspCsv/Target torque
//     TaskCartControl Outputs/CartControl.m_masterCart.m_cartJoints[4].m_motorOutputs/m_cmdMotorEncoder <-> RxPdoMappingCspCsv/Target position
//     TaskCartControl Outputs/CartControl.m_masterCart.m_cartJoints[4].m_motorOutputs/m_controlWord <-> RxPdoMappingCspCsv/Controlword
//     TaskCartControl Outputs/CartControl.m_masterCart.m_cartJoints[4].m_motorOutputs/m_opMode <-> RxPdoMappingCspCsv/Modes of operation
//   MasterController/MasterController Instance <-> MasterController/MasterController Instance
//     TaskArmControl Inputs/MasterArmControl.m_masterInputDataPool.m_cartStatus <-> TaskCartControl Outputs/CartControl.m_cartStatus
//     TaskArmControl Inputs/MasterArmControl.m_masterInputDataPool.m_masterDynaData <-> TaskDynamic Outputs/RobotDynamics.m_masterDynaData
//     TaskArmControl Inputs/MasterArmControl.m_masterInputDataPool.m_safetyData <-> TaskCartControl Outputs/SafetyCheck.m_safetyCheckData
//     TaskDynamic Inputs/RobotDynamics.m_masterJointsData <-> TaskArmControl Outputs/MasterArmControl.m_masterJointsData
//     TaskSafetyCheck Inputs/SafetyCheck.m_cartJointData <-> TaskCartControl Outputs/CartControl.m_cartJointData
//     TaskSafetyCheck Inputs/SafetyCheck.m_cartStatus <-> TaskCartControl Outputs/CartControl.m_cartStatus
//     TaskSafetyCheck Inputs/SafetyCheck.m_masterJointData <-> TaskArmControl Outputs/MasterArmControl.m_masterJointsData
//     TaskSafetyCheck Inputs/SafetyCheck.m_masterStatus <-> TaskArmControl Outputs/MasterArmControl.m_masterStatus

// ---- DUTs/Enum/E_MasterArmState.TcDUT
// Notice: Each state has a corresponding controller, which has a fixed index.
// Add the new state at the end and update the total num
TYPE E_MasterArmState :
(
	MasterArmState_Error := 1,
	MasterArmState_Init :=2,
	MasterArmState_Home :=3,
	MasterArmState_Standby :=4,
	MasterArmState_Matching :=5,
	MasterArmState_Ready :=6,
	MasterArmState_MasterSlave :=7,
	MasterArmState_Clutch :=8,
	MasterArmState_Endoscope :=9,
	MasterArmState_Cart := 10,
	MasterArmState_GravityCali := 11,
	MasterArmState_Test :=12,
	MasterArmState_Disable :=13,
	MasterArmState_Performance :=14,
	MasterArmState_GravityBiasCali :=15,
	
	MasterArmState_totalNum :=MasterArmState_GravityBiasCali
);
END_TYPE

// ---- DUTs/Structure/TasksCommunication/ST_MasterUIData.TcDUT
// Output from UI controller
// Input to master arm control task and cart control task  
TYPE ST_MasterUIData :
STRUCT
	m_motionScale:LREAL := 1.5;
	m_selfCheckFlag:BOOL := FALSE;
	m_masterArmDisableFlag :ARRAY[1..2] OF BOOL:=[2(FALSE)];
	m_enableHandClutch :BOOL :=TRUE;
END_STRUCT
END_TYPE

// ---- DUTs/Structure/TasksCommunication/ST_CartStatus.TcDUT
// Output from cart control task
// Input to master arm control task  
TYPE ST_CartStatus :
STRUCT
	m_initFlag :BOOL:= false;
	m_monitorAngle:LREAL := 0.0;
	m_armSwitch:BOOL := FALSE;
	m_clutchSwitch:BOOL := FALSE;
	m_endoscopeSwitch:BOOL := FALSE;
	m_instrumentPowerSwitch:BOOL := FALSE;
	m_surgonReady :BOOL :=false;
	m_consoleInAdjust:BOOL := FALSE;
	m_monitorInAdjust:BOOL := FALSE;
	m_consoleInManualAdjust:BOOL := FALSE;
	m_ergonAdjustArrival :BOOL;
	m_cancelErgonAdjustArrival :BOOL;
	m_pedalHover : ARRAY [1..2] OF BOOL;
	m_electricKnifePedalTrigger : ARRAY [1..2] OF INT;
END_STRUCT
END_TYPE

// ---- SafetyCheck/safetyCheckDUT/checkDelayTime.TcDUT
TYPE checkDelayTime :
STRUCT
	//motor encoder and joint encoder deviation delay time
	Ti_armJntEncErr:TIME:=T#0.001S;
	//drive error delay time
	Ti_driveErr:TIME:=T#0.1S;
	//joint encoder ununuited delay time
	Ti_linkEncErr:TIME:=T#5S;
	//joint status error delay time 
	Ti_jntStatusErr:TIME:=T#1S;
	//motor current is not update delay time
	Ti_currentIsNotUpdate:TIME:=T#20S;
	//joint postion out of limit
	Ti_outOfLimit:TIME:=T#0.1S;
	//joint follow error delay time
	Ti_armJntFollowErr:TIME:=T#0.1S;
	//joint vel error delay time
	Ti_jntVelErr:TIME:=T#0.05S;
	//joint current error  delay time
	Ti_jntCurrentErr:TIME:=T#0.1S;
	//space pose error  delay time
	Ti_spacePoseErr:TIME:=T#0.1S;

	
	Ti_carDualEncDev:TIME:=T#0.02S;
	Ti_carDriveErr:TIME:=T#1S;
	Ti_carActSec:TIME:=T#10S;
	Ti_carJntStatus:TIME:=T#1S;
	Ti_carTorMotor:TIME:=T#20S;
	Ti_caroutofLimit:TIME:=T#0.1S;
	Ti_carFollowDev:TIME:=T#0.02S;
	Ti_carJntVel:TIME:=T#0.05S;
	Ti_carJntCurrent:TIME:=T#1S;
END_STRUCT
END_TYPE

// ---- GVLs/Arms/GVL_ArmDynamics.TcGVL
{attribute 'global_init_slot' := '49992'}
{attribute 'qualified_only'}
// Robot8 Data
VAR_GLOBAL CONSTANT
	// arm gravity parameters
	(*graParam=[ 2.7244*m3 + 2.7244*m4 + 2.7244*m5 + 2.7244*m6 + 9.8*mx2 + 9.8*mx9,
				9.8*my2 + 9.8*my9,
				3.577*m4 + 3.577*m5 + 3.577*m6 + 0.49*m9 + 9.8*mx3 + 9.8*mx8
				1.5827*m4 + 1.5827*m5 + 1.5827*m6 + 9.8*my3 + 9.8*my8 + 9.8*mz4
				mz5-my4,	my5+mz6,  	mx4,   	mx5, 	mx6,   	my6
				preF2,   k2,   preF3,    k3,    preF5   k5]*)
	g_gravityParam :ARRAY[1..2, 1..16] OF REAL := 
		  [5.2299, -0.0002385, 3.412, 0.9504, -0.03672, 0.02128, 0.0000125, 0.00003509, 0.0001715, -0.01263,
			14.8917, 2220.8492, 10.045, 2875.1933, 3.3359, 630.0, 
		  3.8610, -0.0007155, 3.54376, 1.09147, -0.037617, 0.0236, 0.0000375, 0.00001218, 0.00052255, -0.01313,
			19.53629, 1471.9679, 9.3858, 3100.4051, 2.115, 727.6837];
			
	// gravity deviation
	g_gravityDeviaion :ARRAY[1..2, 1..7] OF REAL :=
	[ 0.0, 0.0, 0.0, 0.0, 0.0, 0.0, 0.0, 
	 0.0, 0.0, 0.0, 0.0, 0.0, 0.0, 0.0];
	  
	// arm friction parameters [a1,b1,...a7,b7];
	// friction = a * gravity + b; only joint 5 and 6 is identified
	g_jntFrictionParam :ARRAY[1..2, 1..14] OF LREAL :=
	[ 0, 0.06026,  0.017, 0.1015,  0.00659, 0.0756,  0.3384, 0.01858,  0.3738, 0.00684, 0.3282, 0.0071,  0, 0.00279,
	  0, 0.0537,  0, 0.0914,  0.0249, 0.07718,  0.298, 0.0334,  0.33139, 0.00768, 0.36325, 0.0076,  0, 0.00254];
	g_maxJntFriction : Vec7d :=[0.2, 0.2, 0.2, 0.1, 0.1, 0.1, 0.01];
	
	//################ dynamic reference model parameters below ###########################
	// link mass [m1, m2, m3, m4, m5, m6, m7, m8, m9]
	g_linkMass :ARRAY[1..9] OF LREAL :=[2.676, 0.825, 0.547, 0.25, 0.195, 0.194, 0.05, 0.111, 0.09] ;
	
	// lin center of amss
	g_linkCOM :ARRAY[1..9,1..3] OF LREAL := [   1.376E-3,    -1.019E-3,  -81.464E-3,
										   90.622E-3,   -0.113E-3,  15.088E-3,
										   167.4E-3,    3.7E-3,     -0.438E-3,
										   0.1E-3,      98.49E-3,   -55.74E-3,
										   0.12E-3,     76.667E-3,  -36E-3,
										   0,           -61.63E-3,  27.3E-3,
										   0.06E-3,     -0.08E-3,   17.671E-3,
										   11E-3,       -3.364E-3,  39.265E-3,
										   143e-3,      0.495e-3,   24.253e-3];
	// link  inertial
    // [Ixx,Iyy,Izz, Ixy,Ixz, Iyz]
 	g_linkInertia :ARRAY[1..9,1..6] OF LREAL :=[  19.63E-3,   16.43E-3,  12.7E-3,   -0.3222E-3,    -0.667E-3,     -0.0268E-3,
												   1.017E-3,   6.637E-3,  5.935E-3,  -0.037E-3,     -0.238E-3,     0.06E-3,
												   0.161E-3,   9.572E-3,  9.586E-3,  0.0447E-3,     0.0277E-3,     0.465E-6,
												   0.992E-3,   0.707E-3,  0.335E-3,  0.2E-6,     2E-6,       0.224E-3,
												   0.402E-3,   0.25E-3,   0.186E-3,  0.002E-6,   -1.2E-6,    0.106E-3,
												   0.281E-3,   0.178E-3,  0.137E-3,  0.076E-6,   0.09E-6,    0.056E-3,
												   0.0255E-3,  0.0259E-3, 5.96E-6,0.34E-6,    -3E-9,      24E-9,
												   0.033E-3,   0.0976E-3, 0.126E-3,  3E-6,       -5E-6,      -0.162E-6,
												   4.9E-6,  0.757E-3,  0.760E-3,  2.6E-6,     -5.3E-6,    -18E-9];

	//################ DO NOT modify parameters below ###########################
	//  motor inertial at link size
	g_motorInertia :ARRAY[1..7] OF LREAL := [34.7E-7, 34.7E-7, 34.7E-7, 9.26E-7, 0.495E-7, 0.495E-7, 0.495E-7];
	
	// spring parameters
	// spring2 [L0, b1, b2, l1, r0]
	g_spring2Param :ARRAY[1..5] OF LREAL :=[114.3E-3, 20E-3, 16E-3, 200E-3, 30E-3];
	// spring3 [L0, b1, b2, l1, r0,d]
	g_spring3Param :ARRAY[1..6] OF LREAL :=[127.5E-3, 20E-3, 23E-3, 200E-3, 32E-3, 23E-3];
	// spring5 [L0, s1, L1, r0, beta]
	g_spring5Param :ARRAY[1..5] OF LREAL :=[70E-3, 17E-3, 121E-3, 7.5E-3, 32.02*g_deg2rad];
	
END_VAR

// ---- GVLs/Arms/GVL_ArmJointCaliData.TcGVL
{attribute 'qualified_only'}
// Robot8 Data-RightArm
VAR_GLOBAL CONSTANT									 
	// absolute encoder value at minimal joint positon
	g_minLinkEncoder :ARRAY[1..g_mArmNum, 1..g_mJntNum] OF DINT :=
		[122745, 128228, 36292, 22430, 20158, 81422, 0,
		 35855, 68924, 4429, 107164, 130111, 42645, 0];
		 
	// absolute encoder value at maximum joint positon
	g_maxLinkEncoder :ARRAY[1..g_mArmNum, 1..g_mJntNum] OF DINT :=
		[36223, 83720, 69818, 109643, 52927, 61070, 0,
		 79841, 24455, 37956, 63571, 31889, 22283, 0];
	
	// absolute encoder value at calibrated positon
	g_caliLinkEncoder :ARRAY[1..g_mArmNum, 1..g_mJntNum] OF DINT :=
		[13120, 107027, 47903, 76302, 102239, 104240, 53627,
		 57523, 46542, 15769, 8255, 81176, 131007, 56205];
	
	 // if absolute encoder value cross zeros within joint motion range
	 // NOTICE: joint 7 is always 0.
	g_linkEncZeroCross :ARRAY[1..g_mArmNum, 1..g_mJntNum] OF INT :=
		[1, 0, 0, 0, 1, 1, 1,
		 0, 0, 0, 1, 0, 1, 1];
		 
	// limit value of gripper hall sensor
	g_minHallSensorValue :ARRAY[1..2] OF DINT:=[8720383,8982527];
	g_maxHallSensorValue :ARRAY[1..2] OF DINT  :=[95684892,94374153];
		 
 	//################ DO NOT modify parameters below ###########################	
	// abolute encoder expanded limit buffer in case there is calibrtion error at limit position
	g_linkEncLimitBuffer : DINT := 1000;
	
	// flag if joint can rotate multiple cycles
	g_multipleCyclesJoint :ARRAY[1..g_mArmNum, 1..g_mJntNum] OF INT :=
		[0, 0, 0, 0, 0, 0, 1,
		 0, 0, 0, 0, 0, 0, 1];
		 
	// joint position at link encoder calibrated point
	g_linkEncCaliJntPos :ARRAY[1..g_mArmNum, 1..g_mJntNum] OF LREAL :=
		[0.0, -PI/2, 0.0, -pi, pi, -PI/2, 0.0,
		 0.0, -PI/2, 0.0, 0.0, pi, PI/2, 0.0];

END_VAR

// ---- GVLs/Arms/GVL_ArmKinematic.TcGVL
// use slot attribute larger than 49990, which is the default one, if it depends on variable in other file
{attribute 'global_init_slot' := '49991'} 
VAR_GLOBAL CONSTANT 

// distance between shoulders of left and right arm
g_shoulderDistance :LREAL := 0.5;

// master arm shoulder rotation in base monitor pose(0 rotate angle)
g_shoulderRotInMonitor : Mat3d :=[0.0,	-1.0,	0.0,
								  0.0,	0.0,	1.0,
								  -1.0,	0.0,	0.0];
 	
(* 
% DH definetion
% !!!!NOTE: q4 is the DH joint position, NOT the motor one
% paramters definiton:
% d1: arm origin to joint1 
% a3: upper arm length
% a4: lower arm length
% d4: wrist height
% a9: parallel structure width
% DH definition:
% index     parent  alpha   a       theta   d       active
% 1         0       0       0       q1      d1      1
% 2         1       -90     0       q2      0       1
% 3         0       0       a3      q3      0       0
% 4         3       -90     a4      q4      d4      1
% 5         4       90      0       q5      0       1
% 6         5       -90     0       q6      0       1
% 7         6       90      0       q7      0       1

% 8         1       -90     0       q8      0       1
% 9         8       0       a9      q9      0       0
% 10        9       0       a3      q10     0       0
% 11        3       0       a9      0       0       fixed

%q4 = motor_q4+q8-q2-90
%q3 = q8 - q2;
%q9 = q2-q8;
%q10 = q8-q2

*)
g_d1:LREAL:=0.26085;
g_d4:LREAL:=0.156;
g_a3:LREAL:=0.278;
g_a4:LREAL:=0.365;
g_a9:LREAL:=0.06;

//alpha,a,d,theta	
g_masterArmDH:ARRAY[1..9,1..4] OF LREAL :=[0,	0,		g_d1,	0,      
										-pi/2,	0,		0,		0,
										0,		g_a3,	0,		0,
										-pi/2,	g_a4,	g_d4,	0,       
										pi/2,	0,		0,		0,
										-pi/2,	0,		0,		0,
										pi/2,	0,		0,		0,
										-pi/2,	0,		0,		0,// joint 8
										0,		g_a9, 	0,		0];
											
// master grip angle fitting coefficients(wrt normalized hall sensor value)
g_masterGripAngleFitCoeff : ARRAY[1..6] OF LREAL :=
	[-2.767665451, 8.744429877, -10.74377687, 6.69841, -2.449592087, 0.5188884865];
g_maxGripAngle : LREAL := 30.0 * g_deg2Rad;
g_minGripAngle :LREAL  := 0.0;

END_VAR

// ---- GVLs/Arms/GVL_ControlParameters.TcGVL
{attribute 'global_init_slot' := '49991'}
VAR_GLOBAL CONSTANT
	// master arm joint position controller parameters
	g_posKp :ARRAY[1..7] OF LREAL :=[50.0,  50.0, 50.0, 4.0, 2.0, 1.0, 0.5];
	g_posKd :ARRAY[1..7] OF LREAL :=[5.0, 2.5, 2.5, 0.1, 0.035, 0.05, 0.01];
	g_posKi :ARRAY[1..7] OF LREAL :=[200.0, 100.0, 100.0, 20.0, 10.0, 10.0, 5.0];
	g_posKiLimit :ARRAY[1..7] OF LREAL :=[500,500,500,500,100,100,100];// define in current
	g_posCtrlLimit :ARRAY[1..7] OF LREAL :=[1000,1000,1000,1000,300,200,200];// define in current
	
	// redundant joint4 following motion parameters
	g_jnt4MaxFollowVel :LREAL :=2*pi;
	g_jnt4MaxFollowAcc :LREAL :=6*pi;
	
	// control tolerance
	g_jntCtrlAngTolLow :LREAL :=0.2*g_deg2Rad;
	g_jntCtrlAngTolHigh :LREAL :=1.0*g_deg2Rad;
	g_cartCtrlPosTol :LREAL :=0.0002;
	g_cartCtrlOriTol :LREAL :=0.2*g_deg2Rad;
	
	// filter cut-off frequency for master grip angle
	g_gripAngLpfCutoffFreq :LREAL := 20;
	
	// filter cut-off frequency for velocity and torque
	g_curJntVelLpfCutoffFreq :LREAL := 30;
	g_cmdJntPosLpfCutoffFreq :LREAL := 30;
	g_curJntTrqLpfCutoffFreq :LREAL := 300;
	g_cmdJntTrqLpfCutoffFreq :LREAL := 300;
	
	// controller would keep command unchanged when error 
	// between command and current value is less than this value
	g_jntCtrlErrForCmdHold :LREAL :=2.0*g_deg2Rad;
	
	// joint is assumed to be static if velocity is less than this value
	g_jntStaticVelThres :LREAL :=0.2*g_deg2Rad;
	
	// home motion parameters
	g_homePosture:ARRAY [1..2, 1..7] OF LREAL:=[0.0, -PI/2, 0, -PI, PI, -PI/2, 0,
							 			  			0.0, -PI/2, 0, 0, PI, PI/2, 0];
	g_homeMaxjntVel:Vec7d:=[1.0, 1.0, 1.0, 1.0, 1.0, 1.0, 1.0];
	g_homeMaxjntAcc:Vec7d:=[1.0, 1.0, 1.0, 2.0, 2.0, 2.0, 2.0];
	g_homeMaxjntJerk:Vec7d:=[7(4.0)];
	
	 // joint observer paramters
	g_jntObvParamL1 :Vec7d :=[0, 0, 0, 0, 300, 300, 0];
	g_jntObvParamL2 :Vec7d :=[0, 0, 0, 0, 1000, 1000, 0];
	g_jntObvParamL3 :Vec7d :=[0, 0, 0, 0, 1000, 1000, 0];
	g_jntObvDamp:Vec7d := [0.8,    0.8,    0.8,     0.05, 0.05, 0.05, 0.05];// TODO: need to be identified
END_VAR

// ---- GVLs/Arms/GVL_ArmJointParameters.TcGVL
{attribute 'global_init_slot' := '49991'}
{attribute 'qualified_only'}
VAR_GLOBAL CONSTANT
	// encoder resolution
	g_incEncoderRes :ARRAY[1..7] OF DINT :=[7(65536)];
	g_absEncoderRes :ARRAY[1..7] OF DINT :=[7(131072)];
	
	// reduction ratio
	g_motorReduction :ARRAY[1..7] OF LREAL :=[115.5/11.5,115.5/11.5,115.5/11.5,(4950.0/190.0)*(22.0/15.0), 2*5625.0/361.0,  2*5625.0/361.0,  2*(66.0/10.0 )];
	g_absEncoderReduction :ARRAY[1..7] OF LREAL :=[7(1.0)];
	
	// motor parameters
	g_motorTrqConst :ARRAY[1..7] OF LREAL :=[0.0385,0.0385,0.0385,0.0299,0.0219,0.0219,0.0219];
	g_motorMaxCurrent :ARRAY[1..7] OF LREAL :=[10.8*1000,10.8*1000,10.8*1000,1.01*1000,314,314,314];//mA
	
	// motor and absEncoder direction
	g_motorDir :ARRAY[1..2, 1..7] OF INT :=[1, -1, 1, -1, 1, -1, -1,	
											1, -1, 1, -1, 1, -1, -1];
	g_asbEncoderDir :ARRAY[1..2, 1..7] OF INT :=[1, -1, 1, 1, -1, 1, 1,
												1, -1, 1, 1, -1, 1, 1];
																 
	// joint position limit
	//TODO: joint7 is given a large limit for initialization moiton
	//NOTE: joint 4 position is coupled with joint 2/3, so the limit is described by link side
	g_minJntPos: ARRAY[1..2,1..7] OF LREAL:=[-60*g_deg2Rad,	-45*g_deg2Rad-pi/2,		-45*g_deg2Rad, 	-pi/2-220*g_deg2Rad, 	-135*g_deg2Rad+pi,		-2.7,		-g_largeNum,
											 -60*g_deg2Rad,	-45*g_deg2Rad-pi/2,		-45*g_deg2Rad,	-pi/2+5*g_deg2Rad,		-135*g_deg2Rad+pi,		-2.7,	-g_largeNum];
	g_maxJntPos: ARRAY[1..2,1..7] OF LREAL:=[60*g_deg2Rad,	60*g_deg2Rad-pi/2,		60*g_deg2Rad,		-pi/2-5*g_deg2Rad,			135*g_deg2Rad+pi,		2.7,		g_largeNum,
								             60*g_deg2Rad,	60*g_deg2Rad-pi/2,		60*g_deg2Rad,		-pi/2+220*g_deg2Rad,			135*g_deg2Rad+pi,		2.7,		g_largeNum];
	
	// joint velocity limit
	g_maxJntVel :ARRAY[1..7] OF LREAL :=[7(2*pi)];
	
END_VAR

// ---- GVLs/Cart/GVL_CartJointCaliData.TcGVL
{attribute 'qualified_only'}
// Robot3 Data
VAR_GLOBAL CONSTANT
	(* cart joints are defiend in sequence as below
	[monitor lift, monitor rotate, armset, pedal] *)

	// absolute encoder value at minimal joint positon
	g_minLinkEncoder :ARRAY[1..4] OF DINT :=[10551943, 13485000, 8646306,11744290];
		 
	// absolute encoder value at maximum joint positon
	g_maxLinkEncoder :ARRAY[1..4] OF DINT :=[9057645, 16376724,7704162,10974938];
	
	// absolute encoder value at calibrated positon
	g_caliLinkEncoder :ARRAY[1..4] OF DINT :=[10551943, 13485000, 8646306,11744290];
	
	// if absolute encoder value cross zeros within joint motion range
	g_linkEncZeroCross :ARRAY[1..4] OF INT :=[0, 0, 0, 0];
		
	 //################ DO NOT modify parameters below ###########################
	// abolute encoder expanded limit buffer in case there is calibrtion error at limit position
	g_linkEncLimitBuffer : DINT := 100000;
	
	// flag if joint can rotate multiple cycles
	g_multipleCyclesJoint :ARRAY[1..4] OF INT :=[0, 0, 0, 0];
		 
	// joint position at link encoder calibrated point
	//TODO: joint2 calibration position need to be checked
	g_linkEncCaliJntPos :ARRAY[1..4] OF LREAL :=[0, 46.264*g_deg2Rad,0,0];

END_VAR

// ---- GVLs/Cart/GVL_CartJointParameters.TcGVL
{attribute 'global_init_slot' := '49991'}
{attribute 'qualified_only'}
VAR_GLOBAL CONSTANT
	(* cart joints are defiend in sequence as below
	[monitor lift, monitor rotate, armset, pedal] *)
	
	// encoder resolution
	g_incEncoderRes :ARRAY[1..4] OF DINT :=[4(65536)];
	g_absEncoderRes :ARRAY[1..4] OF DINT :=[4(16777216)];
	
	// reduction ratio
	g_motorReduction :ARRAY[1..4] OF LREAL :=[2*pi/0.0004682,3317.76,2*pi/0.0004682,1.5*138.0/5*2*pi/0.004];
	// TODO: need to be verified, especially joint2
	g_absEncoderReduction :ARRAY[1..4] OF LREAL :=[1.534, 1 , 1.534, 1.534];// 2*pi/(reduction*g_absEncoderRes)=Line_Resolution_car(from old code, 0.001*2/2^13)
	
	// motor parameters
	g_motorTrqConst :ARRAY[1..4] OF LREAL :=[4(0.0292)];
	g_motorMaxCurrent :ARRAY[1..4] OF LREAL :=[4(1000)];//mA
	
	// motor and absEncoder direction
	g_motorDir :ARRAY[1..4] OF INT :=[1, -1, 1, -1];
	g_asbEncoderDir :ARRAY[1..4] OF INT :=[-1, 1, -1, -1];
																 
	// joint position limit
	g_minJntPos: ARRAY[1..4] OF LREAL:=[0,-31*g_deg2Rad,0,0];
	g_maxJntPos: ARRAY[1..4] OF LREAL:=[0.37,2.61*g_deg2Rad,0.23,0.18];
		
	// joint motion velocity 
	g_jntCtrlMotionVel :ARRAY[1..7] OF LREAL :=[0.015,2*g_deg2Rad,0.01,0.0075];
	

END_VAR

// ---- GVLs/Configs/Robot3/GVL_ArmDynamics_3.TcGVL
{attribute 'global_init_slot' := '49992'}
{attribute 'qualified_only'}
// Robot3 Data
VAR_GLOBAL CONSTANT
	// arm gravity parameters
	(*graParam=[ 2.7244*m3 + 2.7244*m4 + 2.7244*m5 + 2.7244*m6 + 9.8*mx2 + 9.8*mx9,
				9.8*my2 + 9.8*my9,
				3.577*m4 + 3.577*m5 + 3.577*m6 + 0.49*m9 + 9.8*mx3 + 9.8*mx8
				1.5827*m4 + 1.5827*m5 + 1.5827*m6 + 9.8*my3 + 9.8*my8 + 9.8*mz4
				mz5-my4,	my5+mz6,  	mx4,   	mx5, 	mx6,   	my6
				preF2,   k2,   preF3,    k3,    preF5   k5]*)
	g_gravityParam :ARRAY[1..2, 1..16] OF REAL := 
		[ 6.1507, -0.0007155225, 3.320086, 0.48504608, -0.03643, 0.02393, 0.0000375, 0.0000117, 0.00008169, -0.0147358, 
			8.7047302, 3101.998, 7.7845, 1989.9943, 1.112, 477.91541,
		  6.3336386, -0.0002385075, 4.3071, 1.060203, -0.043111496, 0.022730322, 0.0000375, 0.0000117, -0.000929, -0.015102275, 
			7.7845, 3195.0, 12.455128, 2842.287, 2.6162855, 454.267];
			
	// gravity deviation
	g_gravityDeviaion :ARRAY[1..2, 1..7] OF REAL :=
	[ 0.0, 0.0, -0.02, 0.0, 0.0025, 0.005, 0.0, 
	 0.0, 0.0, 0.0, 0.0, -0.0025, -0.005, 0.0];
	  
	// arm friction parameters [a1,b1,...a7,b7];
	// friction = a * gravity + b; only joint 5 and 6 is identified
	g_jntFrictionParam :ARRAY[1..2, 1..14] OF LREAL :=
	[ 0, 0.052118501, 0, 0.050075801, 0.02, 0.036312347, 0.101, 0.02608, 0.21596626, 0.012022009, 0.23862478, 0.004035171, 0, 0.004418365,
	  0, 0.063615008, 0.03, 0.055326576, 0.113, 0.062596658, 0.19, 0.018976863, 0.24246004, 0.0083495406, 0.30998273, 0.0053789188, 0, 0.0046038532];
	g_maxJntFriction : Vec7d :=[0.2, 0.2, 0.2, 0.1, 0.1, 0.1, 0.01];
	
	//################ dynamic reference model parameters below ###########################
	// link mass [m1, m2, m3, m4, m5, m6, m7, m8, m9]
	g_linkMass :ARRAY[1..9] OF LREAL :=[2.676, 0.825, 0.547, 0.25, 0.195, 0.194, 0.05, 0.111, 0.09] ;
	
	// lin center of amss
	g_linkCOM :ARRAY[1..9,1..3] OF LREAL := [   1.376E-3,    -1.019E-3,  -81.464E-3,
										   90.622E-3,   -0.113E-3,  15.088E-3,
										   167.4E-3,    3.7E-3,     -0.438E-3,
										   0.1E-3,      98.49E-3,   -55.74E-3,
										   0.12E-3,     76.667E-3,  -36E-3,
										   0,           -61.63E-3,  27.3E-3,
										   0.06E-3,     -0.08E-3,   17.671E-3,
										   11E-3,       -3.364E-3,  39.265E-3,
										   143e-3,      0.495e-3,   24.253e-3];
	// link  inertial
    // [Ixx,Iyy,Izz, Ixy,Ixz, Iyz]
 	g_linkInertia :ARRAY[1..9,1..6] OF LREAL :=[  19.63E-3,   16.43E-3,  12.7E-3,   -0.3222E-3,    -0.667E-3,     -0.0268E-3,
												   1.017E-3,   6.637E-3,  5.935E-3,  -0.037E-3,     -0.238E-3,     0.06E-3,
												   0.161E-3,   9.572E-3,  9.586E-3,  0.0447E-3,     0.0277E-3,     0.465E-6,
												   0.992E-3,   0.707E-3,  0.335E-3,  0.2E-6,     2E-6,       0.224E-3,
												   0.402E-3,   0.25E-3,   0.186E-3,  0.002E-6,   -1.2E-6,    0.106E-3,
												   0.281E-3,   0.178E-3,  0.137E-3,  0.076E-6,   0.09E-6,    0.056E-3,
												   0.0255E-3,  0.0259E-3, 5.96E-6,0.34E-6,    -3E-9,      24E-9,
												   0.033E-3,   0.0976E-3, 0.126E-3,  3E-6,       -5E-6,      -0.162E-6,
												   4.9E-6,  0.757E-3,  0.760E-3,  2.6E-6,     -5.3E-6,    -18E-9];

	//################ DO NOT modify parameters below ###########################
	//  motor inertial at link size
	g_motorInertia :ARRAY[1..7] OF LREAL := [34.7E-7, 34.7E-7, 34.7E-7, 9.26E-7, 0.495E-7, 0.495E-7, 0.495E-7];
	
	// spring parameters
	// spring2 [L0, b1, b2, l1, r0]
	g_spring2Param :ARRAY[1..5] OF LREAL :=[101.6E-3, 14.5E-3, 15E-3, 172E-3, 31E-3];
	// spring3 [L0, b1, b2, l1, r0,d]
	g_spring3Param :ARRAY[1..6] OF LREAL :=[101.6E-3, 14E-3, 15E-3, 172E-3, 30E-3, 10E-3];
	// spring5 [L0, s1, L1, r0, beta]
	g_spring5Param :ARRAY[1..5] OF LREAL :=[34.93E-3, 34.3E-3, 100E-3, 12.5E-3, 32.02*g_deg2rad];
	
END_VAR

// ---- GVLs/Configs/Robot3/GVL_ArmJointCaliData_3.TcGVL
{attribute 'qualified_only'}
// Robot3 Data
VAR_GLOBAL CONSTANT									 
	// absolute encoder value at minimal joint positon
	g_minLinkEncoder :ARRAY[1..g_mArmNum, 1..g_mJntNum] OF DINT :=
		[5320292, 1637888, 16267012, 9121008, 16329376, 6965264, 0,
		 54048, 5138400, 12480240, 3380960, 9526944, 5270880, 0];
		 
	// absolute encoder value at maximum joint positon
	g_maxLinkEncoder :ARRAY[1..g_mArmNum, 1..g_mJntNum] OF DINT :=
		[16734116, 13586832, 3813732, 14235024, 11133568, 11256240, 0,
		 11534296, 16020072, 96940, 8157232, 13636784, 5270880, 0];
	
	// absolute encoder value at calibrated positon
	g_caliLinkEncoder :ARRAY[1..g_mArmNum, 1..g_mJntNum] OF DINT :=
		[2383568, 16504180, 1109844, 1776208, 6104944, 9165904, 13420592,
		 14507208, 2154776, 14028284, 15460608, 3197104, 7324448, 14964448];
	
	 // if absolute encoder value cross zeros within joint motion range
	 // NOTICE: joint 7 is always 0.
	g_linkEncZeroCross :ARRAY[1..g_mArmNum, 1..g_mJntNum] OF INT :=
		[1, 1, 1, 1, 1, 0, 1,
		 1, 1, 1, 1, 1, 0, 1];
		 
	// limit value of gripper hall sensor
	g_minHallSensorValue :ARRAY[1..2] OF DINT:=[2687067,3145824];
	g_maxHallSensorValue :ARRAY[1..2] OF DINT  :=[34800091,36635182];
		 
 	//################ DO NOT modify parameters below ###########################	
	// abolute encoder expanded limit buffer in case there is calibrtion error at limit position
	g_linkEncLimitBuffer : DINT := 100000;
	
	// flag if joint can rotate multiple cycles
	g_multipleCyclesJoint :ARRAY[1..g_mArmNum, 1..g_mJntNum] OF INT :=
		[0, 0, 0, 0, 0, 0, 1,
		 0, 0, 0, 0, 0, 0, 1];
		 
	// joint position at link encoder calibrated point
	g_linkEncCaliJntPos :ARRAY[1..g_mArmNum, 1..g_mJntNum] OF LREAL :=
		[0.0, -PI/2, 0.0, -pi, pi, -PI/2, 0.0,
		 0.0, -PI/2, 0.0, 0.0, pi, PI/2, 0.0];

END_VAR

// ---- GVLs/GVL_interactUI.TcGVL
{attribute 'qualified_only'}
VAR_GLOBAL
	g_uiParaReload:BOOL:=TRUE;
	
	//true :login；false:logout
	g_userLogged : BOOL;
	
	//master slave scaling : 3:1 , 2:1 , 3:2
	g_masterSlaveScaling : UINT;

	//arm is disable : arm left 1  and  arm right 2
	g_armIsDisbale : UINT;	
	
	//arm assignment method : 1 auto  , 2 manual
	g_armAssignMethod : UINT;
	
	//master arm  mapping  slave arm
	g_armDistributionInfo : ST_arm_distribution;  
	
	//plc definite shutdown
	g_plcPowerOffEnable : BOOL;
	
	//cart in manual adjustment
	g_cartInMotion : BOOL;
	
	//ergonomic control enable 
	g_ergonomicCtrl : ST_ergonCtrlEnable; 
	g_ergonomicCtrlEnableLast : ST_ergonCtrlEnable;
	
	//ergonomic control data
	g_ergonomicCtrlData : ST_ergonomicCtrlData; 

	//ui send reset fault
	g_uiResetFault : UINT;	
	
	//plc send ergonomic current joint position to UI
	g_ergonomicCurData : ST_ergonomicCtrlData;
	
	//head in
	g_surgonHeadIn : BOOL;
	
	//finger clutch on off
	g_fingerClutchOnOff : BOOL;
	
	//error id 
	g_errIdType3 : UDINT;
	g_errIdType2 : UDINT;
	g_errIdType1 : UDINT;
	g_errIdType0 : UDINT;
	
	//master arms and cart self check finshed
	g_masterSelfCheckFinshed : BOOL; 
		
	//PLC version information
	g_plcVersion : STRING := g_SWVersion;

	//stop button ui  : 0 master stop 			
	g_masterStopButton : UINT:=1;
		
	g_digitalZoom : UINT;
	g_hapticZoom : BOOL;
	g_fineTurnning : REAL;
	
	//arm state machine
	g_stateMachineArm1 : INT;
	g_stateMachineArm2 : INT;
	
	// index(0 to 4) of slave arm which is tele-linked to master arm
	g_teleSlaveArm1Idx : INT;
	g_teleSlaveArm2Idx : INT;
	
	//slave check enable  : true start , false end
	g_slaveCheckEnbale : BOOL;

	//0: init status 1: checking 2:check succeed 3: check failed
	g_slaveCheckStatus : UINT;

	//arm switch 
	g_armSwitchEnable : UINT:=0;

	//master hearbeat  : 1s frequency
	g_heartBeat : INT;

	//screen Lock Enable : true Lock  ,  false  unlock
	g_screenLockEnable : BOOL;
END_VAR

// ---- GVLs/GVL_SafetyParameters.TcGVL
{attribute 'global_init_slot' := '49991'}
//TODO: safety check parameters need to be reviewd
VAR_GLOBAL CONSTANT
	
	// safety error counts threshold to trigger fault
	g_faultTriggerCounts :INT :=2;
	
	// arm joint safety error
	g_armMaxJntEncErr :vec7d:=[7(40*g_deg2Rad)];
	g_armMaxJntFollowErr :vec7d:=[7(20*g_deg2Rad)];
	
	// joint limit buffer(outside of joint limit)
	g_armJntPosLimitBuffer :vec7d:=[3(10.0*g_deg2Rad), 4(45.0*g_deg2Rad)];

	//max joint encoder current  saltation
	g_maxJntCurSalta : vec7di:=[7(60000)];
	
	// self check timeout time limit
	g_selfCheckTimeLimit : LREAL:= 15.0;
	
	//arm joint link encoder maximum and minimum values
	g_maxLinkEnc : DINT:=16777215;
	g_minLinkEnc : DINT:=0;
	
	//drive error word
	g_driveErrWord : UDINT:=32;
	
	// master arm cartesion control safety error 
	g_maxCartPosErr :LREAL := 0.005;
	g_maxCartOriErr :LREAL := 5.0*g_deg2Rad;
	

	// master joint safety error
	g_maxJntCtrlErr :LREAL := 15.0*g_deg2Rad;
	g_maxJntEncErr :LREAL := 30.0*g_deg2Rad;
	
	g_minJntPos: ARRAY[1..2,1..7] OF LREAL:=[-60*g_deg2Rad,	-45*g_deg2Rad-pi/2,		-45*g_deg2Rad, 	0, 	-135*g_deg2Rad+pi,		-45*g_deg2Rad-pi/2,		-g_largeNum,
											 -60*g_deg2Rad,	-45*g_deg2Rad-pi/2,		-45*g_deg2Rad,	0,		-135*g_deg2Rad+pi,		-45*g_deg2Rad+pi/2,	-g_largeNum];
	g_maxJntPos: ARRAY[1..2,1..7] OF LREAL:=[60*g_deg2Rad,	60*g_deg2Rad-pi/2,		60*g_deg2Rad,		2*pi,			135*g_deg2Rad+pi,		45*g_deg2Rad-pi/2,		g_largeNum,
								             60*g_deg2Rad,	60*g_deg2Rad-pi/2,		60*g_deg2Rad,		2*pi,			135*g_deg2Rad+pi,		45*g_deg2Rad+pi/2,		g_largeNum];

	
	// cart joint safety error
	g_cartMaxJntCtrlErr :Vec4d := [0.005, 5*g_deg2Rad,0.005, 0.005];
	g_cartMaxJntEncErr :Vec4d :=  [0.005, 5*g_deg2Rad,0.005, 0.005];

	// cart joint limit buffer(outside of joint limit)
	g_cartJntPosLimitBuffer :Vec4d :=[0.05, 10*g_deg2Rad,0.05, 0.05];
	
	// cart joint velocity limit
	g_cartMaxJntVel :Vec4d :=[0.03, 4*g_deg2Rad,0.02,0.015];
	
	// cart joint limit
	g_cartMinJntLimit : Vec4d :=[0-0.1, -(31+5)*g_deg2Rad, 0-0.1, 0-0.1];
	g_cartMaxJntLimit : Vec4d :=[0.38+0.1, (2.6+5)*g_deg2Rad, 0.24+0.1, 0.2+0.1];
	
	//cart joint follow error
	g_cartMaxJntFollowErr : Vec4d :=[0.01, 5*g_deg2rad, 0.01, 0.01];
	
	//cart joint current limit
	g_cartMaxJntCurrent : Vec4d :=[3800*2,3800*2,3800*2,3800*2];
	
	//cart joint encoder detetion value
	g_cartMaxLinkEnc : ARRAY [1..4] OF DINT := [67108863,16777215,67108863,67108863];
	g_cartMinLinkEnc : ARRAY [1..4] OF DINT := [4(0)];
END_VAR

VAR_GLOBAL
	//motor current limit
	g_motorCurrentLimit : Vec7d ;	

	g_arrayErrCodeArm:ARRAY [1..g_maxNum] OF ARRAY [0..100] OF UDINT;	
	g_ArrayErrCodeTypeTest:ARRAY [1..3] OF ARRAY [0..100] OF UDINT;
END_VAR

VAR_GLOBAL CONSTANT
	g_maxNum:INT:=3;
	g_maxArmNum:INT:=2;
	g_maxArmJoint:INT:=7; g_maxCartJoint:INT:=4;
	g_cartNum:UDINT:=3;
	MAX_CSV_ROWS 			: UDINT := 10000;(*最大行数(任务周期为20ms)即10分钟的buffer*)
	MAX_CSV_COLUMNS 		: UDINT := 130;(*最大列数*)
	MAX_CSV_FIELD_LENGTH	: UDINT := 35;(*每个字段的字符长度*)
	MAX_CSV_RING_BUFFER		: UDINT := 3;
	g_ArmNetID: ARRAY[1..g_maxArmNum] OF T_AmsNetId:=['192.168.0.10.4.1','192.168.0.10.9.1'];
	g_JointNetPort:ARRAY[1..g_maxArmNum,1..g_maxArmJoint] OF UINT :=[
											1001,    1002,	1003,	1004,	1005,	1006,	1007,
											1012,    1013,	1014,	1015,	1016,	1017,	1018	];
	g_cartNetID : T_AmsNetId := '192.168.0.10.9.1';
	g_cartJointNetPort:ARRAY[1..g_maxCartJoint] OF UINT :=[1008,    1009,	1010,	1011];
	
END_VAR

// ---- GVLs/GVL_SystemParameters.TcGVL
VAR_GLOBAL CONSTANT
	
	g_SWVersion : STRING := '2(1.0.0.1)';
	
	g_mArmNum :INT := 2;	
	g_mJntNum :INT := 7;	
	g_sArmNum :INT := 4;	
	g_sJntNum :INT := 11;
	g_cartDofs :INT :=6;
	
	
	
	// control loop interval for each task
	g_armCtrlCycleTime :LREAL :=0.00025;
	g_armCtrlFreq :LREAL :=1.0/g_armCtrlCycleTime;
	g_armDynamicCycleTime :LREAL := 0.001;
	g_armDynamicFreq :LREAL := 1.0/g_armDynamicCycleTime;
	g_cartCtrlCycleTime :LREAL := 0.001;
	g_cartCtrlFreq :LREAL := 1.0/g_cartCtrlCycleTime;
	
	// wait time before robot init  for ethercat to stablize 
	g_robotInitWaitTime : LREAL := 1.0;
	g_robotSafetyCheckWaitTime : LREAL :=3.0;
END_VAR

// ---- FBs_BasicControllers/FB_RedunJntControl.TcPOU
// Author: Feijian Ni
// Date: 2023.11.22
FUNCTION_BLOCK FB_RedunJntControl
VAR_INPUT
END_VAR
VAR_OUTPUT
END_VAR
VAR
	// joint 6 deviation from center
	m_jnt6Bias :LREAL;
	
	// max target position step 
	m_maxTargetPosStep :LREAL :=10*g_deg2rad;
	
	// static velocity threshold
	m_staticVelThres :LREAL := 60 *g_deg2Rad;
	
	// static threshold of joint bias
	m_staticBiasThres :LREAL := 30 *g_deg2Rad;
	
	// rudundancy track flag
	m_trackFlag :BOOL;
	
	// joint4 track tolerance
	m_joint4TrackTol :LREAL :=1*g_deg2rad;
	
	// orientation nullspace jacobian
	m_oriNullJaco: Mat4d;
	
	// current manipulation velocity
	m_curManipWVel :LREAL :=0;
	
	// joint4 limit buffer
	m_jntLimitBuffer : LREAL :=2.5*g_deg2Rad;
	
	// control paramters for redundant joint4 position control
//	m_redunJntKp: LREAL:=8.0;
//	m_redunJntKd:LREAL:=0.2;
//	m_redunJntKp: LREAL:=3.0;
//	m_redunJntKd:LREAL:=0.1;
	m_redunJntKp: LREAL:=2.5;
	m_redunJntKd:LREAL:=0.05;
	m_redunJntKi:LREAL:=0;
	m_redunJntKiLimit: LREAL:=200;
	m_redunJntCtrlLimit:LREAL:=1000;

	// max vel and acc for joint4 motion
	m_jnt4MaxFollowVel :LREAL :=2*pi;
	m_jnt4MaxFollowAcc :LREAL :=4*pi;
	m_jnt4MinFollowAcc :LREAL :=1.5*pi;
	m_jnt4MinAccVel:LREAL:= 60 *g_deg2Rad;
	m_jnt4MaxAccVel:LREAL:= 150 *g_deg2Rad;
	
	// max acc scale when approaching joint limit
	m_accScaleNearLimit :LREAL;
	m_maxAccScaleNearLimit :LREAL := 1.0;
	m_accScaleBiasLB :LREAL := 30 *g_deg2Rad;
	m_accScaleBiasUB :LREAL := 45 *g_deg2Rad;

	// final target position of joint4 in motor (not DH , same for below defination) 
	m_jnt4TargetPos: LREAL;
	
	// OTG for joint4 motion
	m_trajFilter :FB_secOrdTrajFilter;
	
	// command joint4 position and veloicty in motor for next cycle
	m_cmdJntPos: LREAL;
	m_cmdJntVel: LREAL;
	m_cmdJntAcc: LREAL;

	// PID for joint position
	m_jntPIDCtrl: FB_PID;
	m_jntCtrlTrq: LREAL;
	
END_VAR

METHOD PROTECTED calcJnt6Bias : LREAL
VAR_IN_OUT CONSTANT
	i_masterArm :FB_MasterArm;
END_VAR
IF 1= i_masterArm.armIdx THEN
	calcJnt6Bias :=i_masterArm.curJntPos[6]+PI/2;
ELSE 
	calcJnt6Bias := i_masterArm.curJntPos[6]-PI/2;
END_IF
END_METHOD

// calculate orientation manipulation velocity(in local coordinate)
METHOD calcManipVel : LREAL
VAR_IN_OUT CONSTANT
	i_masterArm :FB_MasterArm;
END_VAR
VAR
	wVelWrd,wVelLocal:Vec3d;
	rotT:Mat3d;
END_VAR
wVelWrd[1]:= i_masterArm.m_curCartLinkTwist[4];
wVelWrd[2]:= i_masterArm.m_curCartLinkTwist[5];
wVelWrd[3]:= i_masterArm.m_curCartLinkTwist[6];

matTranspose(i_masterArm.curCartPose.m_rot, rotT);
matMultiVec(rotT, wVelWrd, wVelLocal);

wVelLocal[3]:=0;
calcManipVel:=norm(wVelLocal);
END_METHOD

METHOD PROTECTED calcNullJaco : Mat4d;
VAR_IN_OUT CONSTANT
	i_masterArm :FB_MasterArm;
END_VAR
VAR
	i,j:INT;
	oriJaco:Mat34;
	oriJt:Mat43;
	oriJJt:Mat3d;
	oriJJtInv:Mat3d;
	oriJPinv:Mat43;
	JpinvJ :Mat4d;
	eye4d :Mat4d := g_eye4d;
END_VAR
// compute pinv of orientation jacobian
FOR i:=1 TO 3 DO
	FOR j:=1 TO 4 DO
		oriJaco[i,j]:=i_masterArm.simJaco[i+3,j+3];
	END_FOR
END_FOR
matTranspose(oriJaco, oriJt);
matMultiply(oriJaco ,oriJt , oriJJt);
invMat3(oriJJt, oriJJtInv);
matMultiply(oriJt, oriJJtInv, oriJPinv);

// calculate nullspace
matMultiply(oriJPinv, oriJaco, JpinvJ);
matSub(eye4d , JpinvJ, calcNullJaco);
END_METHOD

METHOD PROTECTED calcRedunPos : BOOL
VAR_IN_OUT CONSTANT
	i_masterArm :FB_MasterArm;
END_VAR

VAR 
	j6Bias :LREAL;
	curJntPos : Vec7d;
	jnt4LinkPos, jnt4TargetLinkPos :LREAL;
	singScale:LREAL;
END_VAR
// compute desired joint4 link position
// therotically should be link position, but joint controller use motor pos, so here also use motor pos, or will cause other problems
curJntPos :=  i_masterArm.curJntPos;
jnt4LinkPos:=i_masterArm.jnt4MotorToLink(curJntPos[2],curJntPos[3],curJntPos[4]);

// scale track motion near redundant singularity
IF ABS(m_oriNullJaco[1,1])<g_smallNum THEN
	singScale :=0;
ELSE
	singScale := MAX(ABS(m_oriNullJaco[2,1]/m_oriNullJaco[1,1]), ABS(m_oriNullJaco[3,1]/m_oriNullJaco[1,1]));
END_IF
j6Bias := m_jnt6Bias * ABS(singScale);

j6Bias := LIMIT (-m_maxTargetPosStep, j6Bias, m_maxTargetPosStep);
// final target position
jnt4TargetLinkPos := LIMIT(GVL_ArmJointParameters.g_minJntPos[i_masterArm.armIdx,4]+m_jntLimitBuffer, 
			jnt4LinkPos-j6Bias,GVL_ArmJointParameters.g_maxJntPos[i_masterArm.armIdx,4]-m_jntLimitBuffer); 
			
// convert from link position to motor position
m_jnt4TargetPos:=i_masterArm.jnt4LinkToMotor(curJntPos[2], curJntPos[3], jnt4TargetLinkPos);
END_METHOD

METHOD init : BOOL
VAR_IN_OUT CONSTANT
	i_masterArm :FB_MasterArm;
END_VAR
VAR
	currentRatioMotor2Jnt:LREAL;
END_VAR
m_cmdJntPos:=i_masterArm.curJntPos[4];
m_jnt4TargetPos:=m_cmdJntPos;
m_cmdJntVel:=0;

// init controller
currentRatioMotor2Jnt:=GVL_ArmJointParameters.g_motorTrqConst[4]*GVL_ArmJointParameters.g_motorReduction[4]/1000;
m_jntPIDCtrl.init(g_armCtrlCycleTime,m_redunJntKp,m_redunJntKd,m_redunJntKi,
		m_redunJntKiLimit* currentRatioMotor2Jnt,	m_redunJntCtrlLimit*currentRatioMotor2Jnt);

// init OTG
m_trajFilter.init(m_cmdJntPos,m_cmdJntVel,m_jnt4MaxFollowVel,m_jnt4MaxFollowAcc,g_armCtrlCycleTime);
END_METHOD

METHOD run : LREAL
VAR_IN_OUT CONSTANT
	i_masterArm :FB_MasterArm;
END_VAR
VAR_INPUT
	i_followEnable :BOOL;
END_VAR


VAR
	velScale,limitScale:LREAL;
	maxAcc, minDec:LREAL;
	wVel:Vec3d;

END_VAR
// joint 6 deviation from center
m_jnt6Bias := calcJnt6Bias(i_masterArm);

// calculate nullspace jacobian
m_oriNullJaco := calcNullJaco(i_masterArm);

// calculate manipulation angular velocity(exclude roll velocity)
m_curManipWVel := calcManipVel(i_masterArm);

// check if arm is static
m_trackFlag := startTrackCheck(i_masterArm);

// determin target position of joint4
IF i_followEnable THEN
	// update target redundant joint position
	IF  m_trackFlag THEN
		calcRedunPos(i_masterArm);
	ELSE
		// no control in static state
		IF ABS(m_cmdJntPos-m_jnt4TargetPos)< m_joint4TrackTol THEN
			m_jnt4TargetPos := i_masterArm.curJntPos[4];
			m_cmdJntPos :=i_masterArm.curJntPos[4];
			m_cmdJntVel:=0;
			m_jntPIDCtrl.reset();
			m_trajFilter.init(m_cmdJntPos,m_cmdJntVel,m_jnt4MaxFollowVel,m_jnt4MaxFollowAcc,g_armCtrlCycleTime);
		END_IF
	END_IF
END_IF

// scale following acceleration based on manipulation velocity
velScale := LIMIT (0,(ABS(m_curManipWVel)-m_jnt4MinAccVel)/(m_jnt4MaxAccVel-m_jnt4MinAccVel), 1.0);
maxAcc:=(m_jnt4MaxFollowAcc-m_jnt4MinFollowAcc)*velScale+m_jnt4MinFollowAcc;
//minDec:=m_trajFilter.minDec(m_jnt4TargetPos);
//maxAcc := MAX(maxAcc, minDec);

// scale acceleration when approaching limit
//m_accScaleNearLimit:=1;
limitScale := LIMIT(0.0,(ABS(m_jnt6Bias) - m_accScaleBiasLB)/(m_accScaleBiasUB-m_accScaleBiasLB),1.0);
m_accScaleNearLimit := 1+ limitScale * velScale * m_maxAccScaleNearLimit;
maxAcc:=maxAcc*m_accScaleNearLimit;


// run OTG
m_trajFilter.maxV:=m_curManipWVel;
m_trajFilter.maxA:=maxAcc;
m_trajFilter.run(m_jnt4TargetPos, 0.0, o_cmdAcc=>m_cmdJntAcc,o_cmdVel=>m_cmdJntVel, o_cmdPos=>m_cmdJntPos);

// joint position control torque control
m_jntCtrlTrq:=m_jntPIDCtrl.run(m_cmdJntPos,i_masterArm.curJntPos[4], m_cmdJntVel, i_masterArm.curJntVel[4]);

run:=m_jntCtrlTrq;
END_METHOD

METHOD startTrackCheck : BOOL
VAR_IN_OUT CONSTANT
	i_masterArm :FB_MasterArm;
END_VAR
IF (m_curManipWVel> m_staticVelThres AND i_masterArm.m_curLinkVel[6] * m_jnt6Bias > 0)  OR ABS(m_jnt6Bias)> m_staticBiasThres THEN
	startTrackCheck := TRUE;
ELSE
	startTrackCheck :=FALSE;
END_IF
END_METHOD

END_FUNCTION_BLOCK

// ---- FBs_Robots/FB_MasterArm.TcPOU
FUNCTION_BLOCK FB_MasterArm
VAR
	// arm index, 1 for left arm, 2 for right arm
	m_armIdx: INT;
	
	// grip angle calculator
	m_gripHallSensorIO AT%I* :UDINT;	
	m_gripAngleCalc : FB_GripAngleCalc;
	m_gripAngle :LREAL;
	
	//hand clutch switch IO
	m_handClutchIO AT%I*:UDINT;
	m_handClutchCheck :FB_HandClutchCheck;
	m_handClutchSwitch :BOOL;
	
	// joints
	// NOTICE: all joints are the true active joints, not DH ones!
	m_joints :ARRAY[1..g_mJntNum] OF FB_ArmJoint;
	
	// master gripper roll flip flag, if true, q7 would add pi in FK
	m_gripperRollFlip :BOOL :=False;
	
	// arm cartesian data, defined in each arm origin
	m_curCartPose	:ST_Frame;
	m_curCartTwist: Vec6d;
	m_cmdCartTwist :Vec6d;
	m_cmdCartPose:ST_Frame;
	m_curCartLinkPose :ST_Frame;
	m_curCartLinkTwist :Vec6d;
	
	
	// arm joint data
	m_curMotorPos :Vec7d;
	m_curLinkPos :Vec7d;
	m_curJntPos :Vec7d;
	m_curJntVel :Vec7d;
	m_curLinkVel :Vec7d;
	m_curJntTrq :Vec7d;
	m_rawJntCurrent :Vec7d;
	m_filtJntCurrent :Vec7d;
	m_cmdJntCurrent : Vec7d;
	m_cmdJntTrq :Vec7d;
	m_cmdJntPos :Vec7d;
	m_cmdJntVel :Vec7d;

	
	// arm dynamic data
	m_jntGravity : Vec7d;
	m_jntMassMat : Mat7d;
	m_lambda :Mat6d;
	m_dynaNullspace :Mat7d;
	m_jntFriction :Vec7d;
	m_jntExtTrq :Vec7d;
	m_jntGravityBias :Vec7d;
	
	// arm jacobian 
	m_jaco : Mat67;
	m_linkJaco : Mat67;
	
	// simulated status
	m_simJntPos :Vec7d;
	m_simCartPose : ST_Frame;
	m_simJaco : Mat67;
	
	// joint position controller
	m_jntPIDCtrl :ARRAY[1..g_mJntNum] OF FB_PID;
	
	//joint acceleration
	m_curJntAcc :Vec7d;
	m_curLinkAcc :Vec7d;
END_VAR

PROPERTY armIdx : int
GET
armIdx:=m_armIdx;
END_GET
END_PROPERTY

METHOD PROTECTED calcJaco : BOOL
VAR_IN_OUT CONSTANT
	i_jntPos :ARRAY[1..g_mJntNum] OF LREAL;
END_VAR
VAR_IN_OUT
	r_jaco :ARRAY[1..g_cartDofs, 1..g_mJntNum] OF LREAL;
END_VAR
VAR_INPUT
END_VAR

VAR
	q1,q2, q3, q4, q5, q6, q7 :LREAL;
	d1,d4,a3,a4 :LREAL;
	c1,c2,c3,c4,c5,c6,c7 :LREAL;
	s1,s2,s3,s4,s5,s6,s7 :LREAL;
	c23, s23 :LREAL;
	j:INT;
END_VAR
// !Convert active joint position to DH model for kinematic calculation
q1:=i_jntPos[1];  
q2:=i_jntPos[2];  
q3:=i_jntPos[3]-i_jntPos[2];  //q3=q8-q2
q4:=i_jntPos[4]+i_jntPos[3]-i_jntPos[2]-pi/2;//q4DH=q4motor+q8-q2-90;  
q5:=i_jntPos[5];  
q6:=i_jntPos[6];  
q7:=i_jntPos[7];  
d1:=g_d1;
d4:=g_d4;
a3:=g_a3;
a4:=g_a4;
c1:=COS(q1);
c2:=COS(q2);
c3:=COS(q3);
c4:=COS(q4);
c5:=COS(q5);
c6:=COS(q6);
c7:=COS(q7);
s1:=SIN(q1);
s2:=SIN(q2);
s3:=SIN(q3);
s4:=SIN(q4);
s5:=SIN(q5);
s6:=SIN(q6);
s7:=SIN(q7);
c23:=COS(q2+q3);
s23:=SIN(q2+q3);

// jacobian with DH joints
r_jaco[1,1]:=-s1*(c2*(a3 + a4*c3 - d4*s3) - s2*(d4*c3 + a4*s3)) ;
r_jaco[1,2]:=-c1*(s2*(a3 + a4*c3 - d4*s3) + c2*(d4*c3 + a4*s3)) ;
r_jaco[1,3]:=-c1*(d4*c23 + a4*s23) ;
r_jaco[1,4]:=0 ;
r_jaco[1,5]:=0 ;
r_jaco[1,6]:=0 ;
r_jaco[1,7]:=0;
 
r_jaco[2,1]:=c1*(c2*(a3 + a4*c3 - d4*s3) - s2*(d4*c3 + a4*s3)); 
r_jaco[2,2]:=-s1*(s2*(a3 + a4*c3 - d4*s3) + c2*(d4*c3 + a4*s3)); 
r_jaco[2,3]:=-s1*(d4*c23 + a4*s23); 
r_jaco[2,4]:=0; 
r_jaco[2,5]:=0; 
r_jaco[2,6]:=0; 
r_jaco[2,7]:=0;

 
r_jaco[3,1]:=0 ;
r_jaco[3,2]:=- c1*(c1*c2*(a3 + a4*c3 - d4*s3) - c1*s2*(d4*c3 + a4*s3)) - s1*(c2*s1*(a3 + a4*c3 - d4*s3) - s1*s2*(d4*c3 + a4*s3));
r_jaco[3,3]:=- c1*(a4*c23*c1 - d4*s23*c1) - s1*(a4*c23*s1 - d4*s23*s1);
r_jaco[3,4]:=0;
r_jaco[3,5]:=0;
r_jaco[3,6]:=0 ;
r_jaco[3,7]:=0 ;

r_jaco[4,1]:=0 ;
r_jaco[4,2]:=-s1 ;
r_jaco[4,3]:=-s1 ;
r_jaco[4,4]:=-s23*c1 ;
r_jaco[4,5]:=c23*c1*s4 - c4*s1 ;
r_jaco[4,6]:=- s5*(s1*s4 + c23*c1*c4) - s23*c1*c5 ;
r_jaco[4,7]:=s6*(c5*(s1*s4 + c4*(c1*c2*c3 - c1*s2*s3)) - s5*(c1*c2*s3 + c1*c3*s2)) - c6*(c4*s1 - s4*(c1*c2*c3 - c1*s2*s3));
 
r_jaco[5,1]:=0; 
r_jaco[5,2]:=c1; 
r_jaco[5,3]:=c1; 
r_jaco[5,4]:=-s23*s1; 
r_jaco[5,5]:=c1*c4 + c23*s1*s4; 
r_jaco[5,6]:=s5*(c1*s4 - c23*c4*s1) - s23*c5*s1; 
r_jaco[5,7]:=c6*(c1*c4 - s4*(s1*s2*s3 - c2*c3*s1)) - s6*(c5*(c1*s4 + c4*(s1*s2*s3 - c2*c3*s1)) + s5*(c2*s1*s3 + c3*s1*s2));

r_jaco[6,1]:=1 ;
r_jaco[6,2]:=0 ;
r_jaco[6,3]:=0 ;
r_jaco[6,4]:=-c23 ;
r_jaco[6,5]:=-s23*s4 ;
r_jaco[6,6]:=s23*c4*s5 - c23*c5 ;
r_jaco[6,7]:=- s6*(c23*s5 + s23*c4*c5) - s23*c6*s4;

// jacobian with active joints
// jaco_DH*qdot_DH = jaco_DH * (A * qdot)= jaco * qdot
// A =[ 1  0 0 0 0 0 0
//		0  1 0 0 0 0 0
//		0 -1 1 0 0 0 0
//		0 -1 1 1 0 0 0
//		0 0  0 0 1 0 0
//      0 0  0 0 0 1 0
// 		0 0  0 0 0 0 1]
 FOR j:=1 TO 6 DO 
	 r_jaco[j,2]:=r_jaco[j,2]-r_jaco[j,3]-r_jaco[j,4];
	 r_jaco[j,3]:=r_jaco[j,3]+r_jaco[j,4];
 END_FOR
END_METHOD

PROPERTY cmdCartPose : REFERENCE TO ST_Frame
GET
cmdCartPose REF= m_cmdCartPose;
END_GET
END_PROPERTY

PROPERTY cmdCartTwist : REFERENCE to Vec6d
GET
cmdCartTwist REF= m_cmdCartTwist;
END_GET
END_PROPERTY

PROPERTY cmdJntCurrent :REFERENCE to Vec7d
GET
cmdJntCurrent REF= m_cmdJntCurrent;
END_GET
END_PROPERTY

PROPERTY cmdJntPos : REFERENCE TO Vec7d
GET
cmdJntPos REF= m_cmdJntPos;
END_GET
END_PROPERTY

PROPERTY cmdJntTrq :REFERENCE TO Vec7d
GET
cmdJntTrq REF= m_cmdJntTrq;
END_GET
END_PROPERTY

PROPERTY cmdJntVel : REFERENCE TO Vec7d
GET
cmdJntVel REF= m_cmdJntVel;
END_GET
END_PROPERTY

PROPERTY curCartPose :REFERENCE to ST_Frame
GET
curCartPose REF=m_curCartPose;
END_GET
END_PROPERTY

PROPERTY curCartTwist :REFERENCE TO Vec6d
GET
curCartTwist REF=m_curCartTwist;
END_GET
END_PROPERTY

PROPERTY curJntPos :REFERENCE TO Vec7d
GET
curJntPos REF=m_curJntPos;
END_GET
END_PROPERTY

PROPERTY curJntTrq :REFERENCE TO Vec7d
GET
curJntTrq REF=m_curJntTrq;
END_GET
END_PROPERTY

PROPERTY curJntVel :REFERENCE TO Vec7d
GET
curJntVel REF=m_curJntVel;
END_GET
END_PROPERTY

PROPERTY curLinkPos :REFERENCE TO  Vec7d
GET
curLinkPos REF=m_curLinkPos;
END_GET
END_PROPERTY

PROPERTY curMotorPos :REFERENCE TO Vec7d
GET
curMotorPos REF=m_curMotorPos;
END_GET
END_PROPERTY

PROPERTY PUBLIC dynaNullspace : REFERENCE TO Mat7d
GET
dynaNullspace REF= m_dynaNullspace;
END_GET
END_PROPERTY

METHOD PROTECTED enable : BOOL
VAR_IN_OUT CONSTANT
	i_jntIdx :Vec7i;
END_VAR
VAR
	i :INT ;
END_VAR
FOR i:=1 TO g_mJntNum DO
	IF 1= i_jntIdx[i] THEN
		m_joints[i].enable();
	ELSE
		m_joints[i].disable();
	END_IF
END_FOR
END_METHOD

PROPERTY filtJntCurrent :REFERENCE to Vec7d
GET
filtJntCurrent ref= m_filtJntCurrent;
END_GET
END_PROPERTY

METHOD PUBLIC flipGripper : BOOL
VAR_INPUT
	i_flipFlag :BOOL;
END_VAR
m_gripperRollFlip := i_flipFlag;
END_METHOD

// from active joint position to cartesian pose in arm origin
METHOD PROTECTED forwardKinematic : BOOL
VAR_IN_OUT CONSTANT
	i_jntPos :ARRAY[1..g_mJntNum] OF LREAL;
END_VAR
VAR_IN_OUT
	r_cartPose :ST_Frame;
END_VAR
VAR
	q1,q2, q3, q4, q5, q6, q7 :LREAL;
	d1,d4,a3,a4 :LREAL;
	c1,c2,c3,c4,c5,c6,c7 :LREAL;
	s1,s2,s3,s4,s5,s6,s7 :LREAL;
	c23, s23 :LREAL;
END_VAR
// !Convert active joint position to DH model for kinematic calculation
q1:=i_jntPos[1];  
q2:=i_jntPos[2];  
q3:=i_jntPos[3]-i_jntPos[2];  //q3=q8-q2
q4:=jnt4MotorToLink(i_jntPos[2],i_jntPos[3], i_jntPos[4]);//q4DH=q4motor+q8-q2-90;  
q5:=i_jntPos[5];  
q6:=i_jntPos[6];  
q7:=i_jntPos[7];  

// master roll flip handle
IF m_gripperRollFlip THEN
	q7 := q7+PI;
END_IF

d1:=g_d1;
d4:=g_d4;
a3:=g_a3;
a4:=g_a4;
c1:=COS(q1);
c2:=COS(q2);
c3:=COS(q3);
c4:=COS(q4);
c5:=COS(q5);
c6:=COS(q6);
c7:=COS(q7);
s1:=SIN(q1);
s2:=SIN(q2);
s3:=SIN(q3);
s4:=SIN(q4);
s5:=SIN(q5);
s6:=SIN(q6);
s7:=SIN(q7);
c23:=COS(q2+q3);
s23:=SIN(q2+q3);

// cartesian pose frame
r_cartPose.m_pos[1]:=c1*(a4*c23 - d4*s23 + a3*c2); 
r_cartPose.m_pos[2]:=s1*(a4*c23 - d4*s23 + a3*c2);
r_cartPose.m_pos[3]:=d1 - d4*c23 - a4*s23 - a3*s2;  
r_cartPose.m_rot[1,1]:=c7*(s6*(c4*s1 - s4*(c1*c2*c3 - c1*s2*s3)) + c6*(c5*(s1*s4 + c4*(c1*c2*c3 - c1*s2*s3)) - s5*(c1*c2*s3 + c1*c3*s2))) - s7*(s5*(s1*s4 + c4*(c1*c2*c3 - c1*s2*s3)) + c5*(c1*c2*s3 + c1*c3*s2));
r_cartPose.m_rot[2,1]:=s7*(s5*(c1*s4 + c4*(s1*s2*s3 - c2*c3*s1)) - c5*(c2*s1*s3 + c3*s1*s2)) - c7*(s6*(c1*c4 - s4*(s1*s2*s3 - c2*c3*s1)) + c6*(c5*(c1*s4 + c4*(s1*s2*s3 - c2*c3*s1)) + s5*(c2*s1*s3 + c3*s1*s2)));
r_cartPose.m_rot[3,1]:=- s7*(c23*c5 - s23*c4*s5) - c7*(c23*c6*s5 - s23*s4*s6 + s23*c4*c5*c6); 
r_cartPose.m_rot[1,2]:=- s7*(s6*(c4*s1 - s4*(c1*c2*c3 - c1*s2*s3)) + c6*(c5*(s1*s4 + c4*(c1*c2*c3 - c1*s2*s3)) - s5*(c1*c2*s3 + c1*c3*s2))) - c7*(s5*(s1*s4 + c4*(c1*c2*c3 - c1*s2*s3)) + c5*(c1*c2*s3 + c1*c3*s2)); 
r_cartPose.m_rot[2,2]:=s7*(s6*(c1*c4 - s4*(s1*s2*s3 - c2*c3*s1)) + c6*(c5*(c1*s4 + c4*(s1*s2*s3 - c2*c3*s1)) + s5*(c2*s1*s3 + c3*s1*s2))) + c7*(s5*(c1*s4 + c4*(s1*s2*s3 - c2*c3*s1)) - c5*(c2*s1*s3 + c3*s1*s2)); 
r_cartPose.m_rot[3,2]:=s7*(c23*c6*s5 - s23*s4*s6 + s23*c4*c5*c6) - c7*(c23*c5 - s23*c4*s5); 
r_cartPose.m_rot[1,3]:=s6*(c5*(s1*s4 + c4*(c1*c2*c3 - c1*s2*s3)) - s5*(c1*c2*s3 + c1*c3*s2)) - c6*(c4*s1 - s4*(c1*c2*c3 - c1*s2*s3)); 
r_cartPose.m_rot[2,3]:=c6*(c1*c4 - s4*(s1*s2*s3 - c2*c3*s1)) - s6*(c5*(c1*s4 + c4*(s1*s2*s3 - c2*c3*s1)) + s5*(c2*s1*s3 + c3*s1*s2));
r_cartPose.m_rot[3,3]:=- s6*(c23*s5 + s23*c4*c5) - s23*c6*s4;
END_METHOD

PROPERTY gripAngle : LREAL
GET
gripAngle:=m_gripAngle;
END_GET
END_PROPERTY

PROPERTY gripperRollFlip : BOOL
GET
gripperRollFlip := m_gripperRollFlip;
END_GET
END_PROPERTY

PROPERTY handClutchSwitch : BOOL
GET
handClutchSwitch :=m_handClutchSwitch;
END_GET
END_PROPERTY

METHOD PUBLIC init : BOOL
VAR_INPUT
	i_armIdx:INT;
END_VAR
VAR 
	i :INT ;
	currentRatioMotor2Jnt: LREAL;
END_VAR
// arm statues init
m_armIdx:=i_armIdx;
m_gripAngle:=0;
m_gripAngleCalc.init(m_armIdx);
m_jntGravityBias :=g_zeroVec7d;

// joint init
FOR i:=1 TO g_mJntNum DO
	m_joints[i].init(m_armIdx, i,g_armCtrlCycleTime);
END_FOR

// init joint encoder and position calculation
initJntPos();

// joint controller init
FOR i:=1 TO g_mJntNum DO 
	currentRatioMotor2Jnt:=GVL_ArmJointParameters.g_motorTrqConst[i]*GVL_ArmJointParameters.g_motorReduction[i]/1000;
	m_jntPIDCtrl[i].init(g_armCtrlCycleTime,g_posKp[i],g_posKd[i],g_posKi[i],
		g_posKiLimit[i]* currentRatioMotor2Jnt,	g_posCtrlLimit[i]*currentRatioMotor2Jnt);
END_FOR
END_METHOD

METHOD public initJntPos : BOOL
VAR_INPUT
END_VAR
VAR
	i:INT ;
	initLinkPos:LREAL;
END_VAR
// joint init
FOR i:=1 TO g_mJntNum DO
	m_joints[i].initJntPos();
END_FOR

// link position of joint4 is influenced by joint2 and joint3, need to handle seperately
initLinkPos:=jnt4LinkToMotor(m_joints[2].initLinkPos,m_joints[3].initLinkPos, m_joints[4].initLinkPos);
m_joints[4].initJntPosReset(initLinkPos);

// update arm status after joint position is re-init
updateStatus();
END_METHOD

// from cartesian pose in arm origin to active joint position
METHOD PROTECTED inverseKinematic : BOOL
VAR_INPUT
	q4:LREAL;
	solution_ID:INT;
END_VAR
VAR_IN_OUT CONSTANT
	i_curCartPose :ST_Frame;
END_VAR
VAR_IN_OUT
	r_jntPos :ARRAY[1..g_mJntNum] OF LREAL;
END_VAR
VAR
	a3,a4,d1,d4:LREAL;
	px,py,pz:lreal;
	nx,ny,nz:lreal;
	ox,oy,oz:lreal;
	ax,ay,az:lreal;

	q1,q2,q3,q5,q6,q7:LREAL;
	
	q11,q12:LREAL;
	k1,A,B,C,fi,R0,q21,q22:lreal;
	ins1,ins2:lreal;
	
	A11,A12,A21,A22,C1,C2:lreal;
	SIN23,COS23,q23:lreal;
	
	T_74_left_23,q61,q62:lreal;
	T_74_left_13,T_74_left_33:lreal;
	T_74_left_21,T_74_left_22:LREAL;	
	
	succeed_1,succeed_2,succeed:BOOL;
END_VAR


//***********************单臂逆向运动学**************************//
d1:=g_d1;
d4:=g_d4;
a3:=g_a3;
a4:=g_a4;

nx:=i_curCartPose.m_rot[1,1];  ny:=i_curCartPose.m_rot[2,1];  nz:=i_curCartPose.m_rot[3,1];
ox:=i_curCartPose.m_rot[1,2]; oy:=i_curCartPose.m_rot[2,2];  oz:=i_curCartPose.m_rot[3,2];
ax:=i_curCartPose.m_rot[1,3];  ay:=i_curCartPose.m_rot[2,3];  az:=i_curCartPose.m_rot[3,3];
px:=i_curCartPose.m_pos[1]; py:=i_curCartPose.m_pos[2]; pz:=i_curCartPose.m_pos[3];


//求解q1
q11:=atan2(y:= py, x:= px);
q12:=-q11;
IF (Solution_ID<=4) THEN
	q1:=q11;
ELSE
	q1:=q12;
END_IF



//求解q2
k1:=px*COS(q1) + py*SIN(q1);
A:=2*a3*pz - 2*a3*d1;
B:=2*a3*k1;
C:=a3*a3 - a4*a4 + d1*d1 - 2*d1*pz - d4*d4 + k1*k1 + pz*pz;
fi:=atan2(y:= B, x:= A);

R0:=SQRT(A*A+B*B);

//*************程序保护性处理，避免软件崩溃***************//
IF ABS(C/R0)>1 THEN
	succeed_1:=FALSE;
	succeed:=FALSE;
	RETURN;
ELSE
	succeed_1:=TRUE;
END_IF

ins1:=atan2(y:= C/R0, x:= SQRT(1-(C/R0)*(C/R0)));
q21:=fi-ins1;
ins2:=atan2(y:= C/R0, x:= -SQRT(1-(C/R0)*(C/R0)));
q22:=fi-ins2;

IF (Solution_ID=1) OR (Solution_ID=2) OR (Solution_ID=5) OR (Solution_ID=6) THEN
	q2:=q21;
ELSE
	q2:=q22;
END_IF




//求解q3
A11:=- d4;
A12:=a4;
A21:=- a4;
A22:=-d4;
C1:=k1- a3*COS(q2);
C2:=pz - d1 + a3*SIN(q2);
sin23:=(C1*A22-C2*A12)/(A11*A22-A21*A12);
cos23:=(C2*A11-C1*A21)/(A11*A22-A21*A12);
q23:=atan2(y:= sin23, x:= cos23);
q3:=q23-q2;




//求解q6
T_74_left_23:=ax*(COS(q4)*SIN(q1) - COS(q1)*COS(q2)*COS(q3)*SIN(q4) + COS(q1)*SIN(q2)*SIN(q3)*SIN(q4)) - ay*(COS(q1)*COS(q4) + COS(q2)*COS(q3)*SIN(q1)*SIN(q4) - SIN(q1)*SIN(q2)*SIN(q3)*SIN(q4)) + az*SIN(q2 + q3)*SIN(q4);

//*************程序保护性处理，避免软件崩溃***************//
IF ABS(T_74_left_23>1) THEN
	succeed_2:=FALSE;
	succeed:=FALSE;
	RETURN;
ELSE
	succeed_2:=TRUE;
END_IF

q61:=ACOS(-T_74_left_23);
q62:=-ACOS(-T_74_left_23);
IF (Solution_ID=1) OR (Solution_ID=3) OR (Solution_ID=5) OR (Solution_ID=7) THEN
	q6:=q61;
ELSE
	q6:=q62;
END_IF


//求解q5
T_74_left_13:=ax*(SIN(q1)*SIN(q4) + COS(q1)*COS(q2)*COS(q3)*COS(q4) - COS(q1)*COS(q4)*SIN(q2)*SIN(q3)) - ay*(COS(q1)*SIN(q4) - COS(q2)*COS(q3)*COS(q4)*SIN(q1) + COS(q4)*SIN(q1)*SIN(q2)*SIN(q3)) - az*SIN(q2 + q3)*COS(q4);
T_74_left_33:=- az*COS(q2 + q3) - ax*SIN(q2 + q3)*COS(q1) - ay*SIN(q2 + q3)*SIN(q1);
q5:=atan2(y:= T_74_left_33*SIN(q6), x:= T_74_left_13*SIN(q6));


//求解q7
T_74_left_21:=nx*(COS(q4)*SIN(q1) - COS(q1)*COS(q2)*COS(q3)*SIN(q4) + COS(q1)*SIN(q2)*SIN(q3)*SIN(q4)) - ny*(COS(q1)*COS(q4) + COS(q2)*COS(q3)*SIN(q1)*SIN(q4) - SIN(q1)*SIN(q2)*SIN(q3)*SIN(q4)) + nz*SIN(q2 + q3)*SIN(q4);
T_74_left_22:=ox*(COS(q4)*SIN(q1) - COS(q1)*COS(q2)*COS(q3)*SIN(q4) + COS(q1)*SIN(q2)*SIN(q3)*SIN(q4)) - oy*(COS(q1)*COS(q4) + COS(q2)*COS(q3)*SIN(q1)*SIN(q4) - SIN(q1)*SIN(q2)*SIN(q3)*SIN(q4)) + oz*SIN(q2 + q3)*SIN(q4);
q7:=atan2(y:= -T_74_left_22*SIN(q6), x:= T_74_left_21*SIN(q6));


//! convert DH joint postion to active joint position
r_jntPos[1]:=q1;
r_jntPos[2]:=q2;
r_jntPos[3]:=q3+q2; // q8 = q3+q2
r_jntPos[4]:=q4+q2-r_jntPos[3]+pi/2;//q4DH=q4motor+q8-q2-90;  
r_jntPos[5]:=q5;
r_jntPos[6]:=q6;
r_jntPos[7]:=q7;

succeed:=TRUE;
inverseKinematic:=succeed;
END_METHOD

METHOD PUBLIC isEnabled : BOOL
VAR_IN_OUT CONSTANT
	i_jntIdx :Vec7i;
END_VAR
VAR
	i :INT ;
END_VAR
isEnabled := TRUE;
FOR i:=1 TO g_mJntNum DO
	IF 1= i_jntIdx[i] THEN
		isEnabled :=  (m_joints[i].isEnabled() AND isEnabled);
	END_IF
END_FOR
END_METHOD

PROPERTY jaco :REFERENCE to Mat67
GET
jaco ref= m_jaco;
END_GET
END_PROPERTY

//convert joint4 position from link side to motor side
METHOD PUBLIC jnt4LinkToMotor : LREAL
VAR_INPUT
	i_q2 :LREAL;
	i_q3:LREAL;
	i_q4Link :LREAL;
END_VAR
jnt4LinkToMotor:=i_q4Link-i_q3+i_q2+pi/2;//q4motor=q4DH-q8+q2+90;
END_METHOD

//convert joint4 position from motor side to link side
METHOD public jnt4MotorToLink : LREAL
VAR_INPUT
	i_q2 :LREAL;
	i_q3:LREAL;
	i_q4Motor :LREAL;
END_VAR
jnt4MotorToLink:=i_q4Motor+i_q3-i_q2-pi/2;//q4DH=q4motor+q8-q2-90;
END_METHOD

PROPERTY jntExtTrq :REFERENCE TO Vec7d
GET
jntExtTrq REF= m_jntExtTrq;
END_GET
END_PROPERTY

PROPERTY jntFriction :REFERENCE TO Vec7d
GET
jntFriction REF= m_jntFriction;
END_GET
END_PROPERTY

PROPERTY jntGravity :REFERENCE to Vec7d
GET
jntGravity ref=m_jntGravity;
END_GET
END_PROPERTY

PROPERTY jntGravityBias :REFERENCE to Vec7d
GET
jntGravityBias ref=m_jntGravityBias;
END_GET
SET // PUBLIC
m_jntGravityBias := jntGravityBias;
END_SET
END_PROPERTY

PROPERTY PUBLIC massMat :REFERENCE to Mat7d
GET
massMat ref=m_jntMassMat;
END_GET
END_PROPERTY

PROPERTY rawJntCurrent :REFERENCE to Vec7d
GET
rawJntCurrent ref=m_rawJntCurrent;
END_GET
END_PROPERTY

PROPERTY simCartPose :REFERENCE to ST_Frame
GET
simCartPose REF=m_simCartPose;
END_GET
END_PROPERTY

PROPERTY simJaco :REFERENCE TO mat67
GET
simJaco REF=m_simJaco;
END_GET
END_PROPERTY

// update joints control command
METHOD PUBLIC updateCmds : BOOL
VAR_IN_OUT CONSTANT
	i_armCtrlCmd : ST_ArmCtrlCmds;
END_VAR
VAR
	i:INT;
END_VAR
m_cmdJntTrq:=i_armCtrlCmd.m_cmdJntTrq;
m_cmdJntPos :=i_armCtrlCmd.m_cmdJntPos;
m_cmdJntVel :=i_armCtrlCmd.m_cmdJntVel;
m_cmdCartTwist := i_armCtrlCmd.m_cmdCartTwist;
m_cmdCartPose :=i_armCtrlCmd.m_cmdCartPose;
m_simJntPos:=i_armCtrlCmd.m_cmdJntPos;

// update simulated master arm
updateSimStatus();

// enable/disable joints
enable(i_armCtrlCmd.m_jntEnableFlag);

// position/torque control
FOR i:=1 TO g_mJntNum DO 
	IF i_armCtrlCmd.m_jntOPMode[i]=DriverOPMode_PosTrq THEN
		// position controller and gravity feedforward
		m_cmdJntTrq[i]:=m_jntPIDCtrl[i].run(i_armCtrlCmd.m_cmdJntPos[i],m_curJntPos[i],i_armCtrlCmd.m_cmdJntVel[i],m_curJntVel[i]);
		m_cmdJntTrq[i]:=m_cmdJntTrq[i]+m_jntGravity[i];
		m_joints[i].updateCmds(DriverOPMode_Trq,i_armCtrlCmd.m_cmdJntPos[i],m_cmdJntTrq[i]);
	ELSIF i_armCtrlCmd.m_jntOPMode[i]=DriverOPMode_Trq THEN
		// gravity feedforward
		m_jntPIDCtrl[i].reset();
		m_cmdJntTrq[i]:=m_cmdJntTrq[i]+m_jntGravity[i] + m_jntGravityBias[i];
		m_joints[i].updateCmds(DriverOPMode_Trq,i_armCtrlCmd.m_cmdJntPos[i],m_cmdJntTrq[i]);
	ELSE
		m_jntPIDCtrl[i].reset();
		m_cmdJntTrq[i]:=0;
		m_joints[i].updateCmds(DriverOPMode_Pos,i_armCtrlCmd.m_cmdJntPos[i],m_cmdJntTrq[i]);
	END_IF
	
END_FOR
END_METHOD

METHOD PUBLIC updateDyna : BOOL
VAR_IN_out constant
	masterDynaData : ST_MasterDynaData;
END_VAR
m_jntMassMat:=masterDynaData.m_massMat[m_armIdx];
m_lambda:=masterDynaData.m_lambda[m_armIdx];
m_dynaNullspace:=masterDynaData.m_dynaNullspace[m_armIdx];
m_jntGravity:=masterDynaData.m_gravity[m_armIdx];
m_jntFriction:=masterDynaData.m_friction[m_armIdx];
m_jntExtTrq := masterDynaData.m_jntExtTrq[m_armIdx];
END_METHOD

METHOD PUBLIC updateSimStatus : BOOL
VAR_INPUT
END_VAR
// simulated cartesion pose 
forwardKinematic(m_simJntPos,m_simCartPose);

// simulated jacobian
calcJaco(m_simJntPos,m_simJaco);
END_METHOD

// update arm status, including kinematic and dynamic
METHOD PUBLIC updateStatus : BOOL
VAR_INPUT
END_VAR
VAR 
	i,j:INT;
END_VAR
// grip angle
m_gripAngle :=m_gripAngleCalc.run(m_gripHallSensorIO);

// check hand clutch
m_handClutchSwitch :=  m_handClutchCheck.run(m_handClutchIO);

// update joint data
FOR i:=1 TO g_mJntNum DO
	m_joints[i].updateStatus();
END_FOR

// get joint data
FOR i:=1 TO g_mJntNum DO
	m_curMotorPos[i]:=m_joints[i].motorPos;
	m_curLinkPos[i]:=m_joints[i].linkPos;
	m_curJntPos[i]:=m_joints[i].jntPos;
	m_curJntVel[i]:=m_joints[i].jntVel;
	m_curLinkVel[i] := m_joints[i].m_curLinkVel;	
	m_curJntAcc[i]:=m_joints[i].m_curJntAcc;
	m_curLinkAcc[i]:=m_joints[i].m_curLinkAcc;	
	m_curJntTrq[i]:=m_joints[i].jntTrq;
	m_rawJntCurrent[i]:=m_joints[i].rawCurrent;
	m_filtJntCurrent[i]:=m_joints[i].filtCurrent;
	m_cmdJntCurrent[i]:=m_joints[i].cmdCurrent;
END_FOR 
m_curLinkPos[4]:=jnt4LinkToMotor(m_curLinkPos[2],m_curLinkPos[3], m_curLinkPos[4]);// q4motor=q4DH-q8+q2+90; 
m_curLinkVel[4]:= m_curLinkVel[4] - m_curLinkVel[3] + m_curLinkVel[2]; 
m_curLinkAcc[4]:= m_curLinkAcc[4] - m_curLinkAcc[3] + m_curLinkAcc[2];

// cartesion pose
forwardKinematic(m_curJntPos,m_curCartPose);
forwardKinematic(m_curLinkPos,m_curCartLinkPose);

// jacobian
calcJaco(m_curJntPos,m_jaco);
calcJaco(m_curLinkPos,m_linkJaco);

// cartesian twist
matMultiVec(m_jaco,m_curJntVel,m_curCartTwist);
matMultiVec(m_linkJaco,m_curLinkVel,m_curCartLinkTwist);
END_METHOD

END_FUNCTION_BLOCK

// ---- FBs_Robots/FB_ArmJoint.TcPOU
FUNCTION_BLOCK FB_ArmJoint EXTENDS FB_JointBase
VAR_INPUT
END_VAR
VAR_OUTPUT
END_VAR
VAR
END_VAR

METHOD PUBLIC init : BOOL
VAR_INPUT
	i_armIdx :INT;
	i_jntIdx :INT;
	i_controlCycleTime :LREAL;
END_VAR
m_cycleTime := i_controlCycleTime;

// hardware parameters
m_motorEncoderRes :=GVL_ArmJointParameters.g_incEncoderRes[i_jntIdx];
m_linkEncoderRes :=GVL_ArmJointParameters.g_absEncoderRes[i_jntIdx];
m_motorReduction :=GVL_ArmJointParameters.g_motorReduction[i_jntIdx];
m_linkEncoderReduction :=GVL_ArmJointParameters.g_absEncoderReduction[i_jntIdx];
m_trqConst :=GVL_ArmJointParameters.g_motorTrqConst[i_jntIdx];
m_maxCurrent :=GVL_ArmJointParameters.g_motorMaxCurrent[i_jntIdx];
m_motorDir :=GVL_ArmJointParameters.g_motorDir[i_armIdx,i_jntIdx];								
m_linkEncoderDir :=GVL_ArmJointParameters.g_asbEncoderDir[i_armIdx,i_jntIdx];
m_minJntPos	:=GVL_ArmJointParameters.g_minJntPos[i_armIdx,i_jntIdx];
m_maxJntPos	:=GVL_ArmJointParameters.g_maxJntPos[i_armIdx,i_jntIdx];

//link encoder calibartion data
m_minLinkEncoder :=GVL_ArmJointCaliData.g_minLinkEncoder[i_armIdx, i_jntIdx] - m_linkEncoderDir*GVL_ArmJointCaliData.g_linkEncLimitBuffer; // expand limit
m_maxLinkEncoder :=GVL_ArmJointCaliData.g_maxLinkEncoder[i_armIdx, i_jntIdx] + m_linkEncoderDir*GVL_ArmJointCaliData.g_linkEncLimitBuffer; // expand limit
m_caliLinkEncoder :=GVL_ArmJointCaliData.g_caliLinkEncoder[i_armIdx, i_jntIdx];
m_linkEncCaliJntPos :=GVL_ArmJointCaliData.g_linkEncCaliJntPos[i_armIdx, i_jntIdx];
m_linkEncZeroCross :=GVL_ArmJointCaliData.g_linkEncZeroCross[i_armIdx, i_jntIdx];
m_multiCycles :=GVL_ArmJointCaliData.g_multipleCyclesJoint[i_armIdx,i_jntIdx];

// convert cali link encoder if joint cross zero
IF 1=m_linkEncZeroCross THEN
	IF 1=m_linkEncoderDir AND m_caliLinkEncoder < m_minLinkEncoder THEN
		m_caliLinkEncoder := GVL_ArmJointCaliData.g_caliLinkEncoder[i_armIdx, i_jntIdx] + m_linkEncoderRes;
	ELSIF -1=m_linkEncoderDir AND m_caliLinkEncoder < m_maxLinkEncoder THEN
		m_caliLinkEncoder := GVL_ArmJointCaliData.g_caliLinkEncoder[i_armIdx, i_jntIdx] + m_linkEncoderRes;
	END_IF
END_IF

// macro data
m_trq2CurrentRatio:=m_motorDir * 1000.0/(m_trqConst*m_motorReduction);
m_current2TrqRatio:=m_motorDir * (m_trqConst*m_motorReduction)/1000.0;
m_linkEnc2PosRatio := 2*PI*m_linkEncoderDir/(m_linkEncoderReduction*m_linkEncoderRes);
m_motorEnc2PosRatio := 2*PI * m_motorDir/(m_motorReduction * m_motorEncoderRes);

// motor data init
m_curJntVel:=0;
m_curJntTrq :=0;
m_rawCurrent :=0;
m_filtCurrent :=0;
m_cmdJntVel :=0.0;
m_cmdJntTrq :=0.0;
m_cmdCurrent := 0.0;

// filter init
m_jntVelLpf.init(1, g_curJntVelLpfCutoffFreq, g_armCtrlFreq);
m_linkVelLpf.init(1, g_curJntVelLpfCutoffFreq, g_armCtrlFreq);
m_jntAccLpf.init(1, g_curJntVelLpfCutoffFreq*0.2, g_armCtrlFreq); 
m_linkAccLpf.init(1, g_curJntVelLpfCutoffFreq*0.2, g_armCtrlFreq); 
m_cmdTrqLpf.init(1, g_cmdJntTrqLpfCutoffFreq, g_armCtrlFreq);
m_curTrqLpf.init(1, g_curJntTrqLpfCutoffFreq, g_armCtrlFreq);


// driver init value
m_motorOutputs.m_controlWord:=DriverCtrlWord_INIT;
m_motorOutputs.m_opMode:=INT_TO_SINT(DriverOPMode_Pos);
m_motorOutputs.m_cmdCurrent:=0;
m_motorOutputs.m_cmdMotorEncoder:=m_motorInputs.m_motorEncoder;
END_METHOD

END_FUNCTION_BLOCK

// ---- FBs_Robots/FB_JointBase.TcPOU
FUNCTION_BLOCK FB_JointBase
VAR
	// motor IO
	m_motorInputs AT%I*	:ST_MotorInputs;
	m_motorOutputs AT%Q* :ST_MotorOutputs;
		
	// cycle time
	m_cycleTime :LREAL;
	
	// calibrated link encoder data
	m_minLinkEncoder :DINT;
	m_maxLinkEncoder :DINT;
	m_caliLinkEncoder :DINT;
	m_linkEncCaliJntPos :LREAL;
	m_linkEncZeroCross :INT;
	m_initMotorEnc : DINT;
	m_multiCycles :INT;
	
	// joint position from link encoder after power on
	m_initLinkPos :LREAL;
	
	// data for link encoder multiple cycles
	m_lastLinkEncoder :DINT;
	m_linkEncCycles:INT;
	
	// device paramters
	m_motorEncoderRes :DINT;
	m_linkEncoderRes :DINT;
	m_motorReduction :LREAL;
	m_linkEncoderReduction :LREAL;
	m_trqConst :LREAL;
	m_maxCurrent :LREAL;
	m_motorDir :INT;								
	m_linkEncoderDir :INT;
	m_minJntPos: LREAL;
	m_maxJntPos: LREAL;
	
	// macro defined data for quick calculation
	m_trq2CurrentRatio:LREAL;
	m_current2TrqRatio:LREAL;
	m_linkEnc2PosRatio :LREAL;
	m_motorEnc2PosRatio :LREAL;
	
	// joint data
	m_curMotorPos :LREAL;
	m_curLinkPos :LREAL;
	m_curJntPos	:LREAL;
	m_curJntVel :LREAL;
	m_curLinkVel :LREAL;
	m_curJntTrq :	LREAL;
	m_rawCurrent : LREAL;
	m_filtCurrent : LREAL;
	m_cmdJntPos :LREAL;
	m_cmdJntVel :LREAL;
	m_cmdJntTrq :LREAL;
	m_cmdCurrent : LREAL;
	m_lastJntPos :LREAL;
	m_lastLinkPos: LREAL;
	
	// velocity filter
	m_jntVelLpf :FB_LowPassFilter;
	m_linkVelLpf :FB_LowPassFilter;
	
	// current and command torque filter
	m_curTrqLpf : FB_LowPassFilter;
	m_cmdTrqLpf :FB_LowPassFilter;
	
	//joint acceleration and filter
	m_curJntAcc :LREAL;
	m_curLinkAcc:LREAL;
	m_lastJntVel: LREAL;
	m_lastLinkVel: LREAL;
	m_jntAccLpf :FB_LowPassFilter;
	m_linkAccLpf :FB_LowPassFilter;
END_VAR

PROPERTY cmdCurrent : LREAL
GET
cmdCurrent:=m_cmdCurrent;
END_GET
END_PROPERTY

METHOD PUBLIC disable : BOOL
VAR_INPUT
END_VAR
m_motorOutputs.m_controlWord:=DriverCtrlWord_INIT;
disable:=true;
END_METHOD

METHOD PUBLIC enable : BOOL
VAR_INPUT
END_VAR
IF DriverStatusWord_INIT = m_motorInputs.m_statusWord THEN
	m_motorOutputs.m_controlWord:=DriverCtrlWord_PREOP;
	enable := FALSE;
ELSIF DriverStatusWord_PREOP = m_motorInputs.m_statusWord THEN
	m_motorOutputs.m_controlWord:=DriverCtrlWord_OP;
	enable :=  FALSE;
ELSIF DriverStatusWord_OP = m_motorInputs.m_statusWord THEN
	enable :=  TRUE;
//ELSE
//	m_motorOutputs.m_controlWord:=DriverCtrlWord_INIT;
//	enable :=  FALSE;
END_IF
END_METHOD

PROPERTY filtCurrent : LREAL
GET
filtCurrent:=m_filtCurrent;
END_GET
END_PROPERTY

